C07196=1037.272,370.437,-131.137,172.942,44.628,158.763
C07197=1037.264,370.189,-131.097,172.935,44.625,158.762
C07198=1037.256,369.942,-131.057,172.928,44.622,158.760
C07199=1037.248,369.696,-131.017,172.921,44.619,158.759
C07200=1037.240,369.449,-130.977,172.914,44.615,158.757
C07201=1037.231,369.203,-130.937,172.907,44.612,158.756
C07202=1037.223,368.957,-130.897,172.900,44.608,158.754
C07203=1037.215,368.710,-130.857,172.894,44.605,158.753
C07204=1037.207,368.462,-130.817,172.887,44.602,158.751
C07205=1037.198,368.216,-130.778,172.881,44.599,158.750
C07206=1037.190,367.969,-130.739,172.874,44.595,158.748
C07207=1037.182,367.723,-130.698,172.867,44.592,158.747
C07208=1037.173,367.476,-130.659,172.860,44.589,158.745
C07209=1037.166,367.229,-130.619,172.853,44.586,158.744
C07210=1037.157,366.983,-130.579,172.848,44.582,158.743
C07211=1037.149,366.736,-130.539,172.841,44.579,158.741
C07212=1037.141,366.489,-130.500,172.834,44.576,158.740
C07213=1037.132,366.243,-130.461,172.827,44.573,158.738
C07214=1037.125,365.996,-130.421,172.820,44.570,158.737
C07215=1037.116,365.749,-130.382,172.814,44.566,158.735
C07216=1037.109,365.502,-130.342,172.807,44.563,158.734
C07217=1037.101,365.256,-130.303,172.801,44.560,158.733
C07218=1037.093,365.009,-130.263,172.794,44.557,158.731
C07219=1037.085,364.762,-130.224,172.788,44.554,158.730
C07220=1037.076,364.516,-130.185,172.781,44.551,158.728
C07221=1037.069,364.269,-130.145,172.774,44.548,158.727
C07222=1037.056,363.891,-130.084,172.765,44.543,158.725
C07223=1037.044,363.513,-130.025,172.755,44.538,158.723
C07224=1037.032,363.134,-129.964,172.745,44.533,158.721
C07225=1037.020,362.756,-129.904,172.735,44.528,158.719
C07226=1037.012,362.510,-129.865,172.729,44.525,158.717
C07227=1037.004,362.262,-129.826,172.722,44.522,158.716
C07228=1036.996,362.015,-129.786,172.716,44.519,158.715
C07229=1036.988,361.769,-129.748,172.710,44.516,158.713
C07230=1036.981,361.522,-129.708,172.703,44.513,158.712
C07231=1036.972,361.275,-129.669,172.697,44.510,158.711
C07232=1036.964,361.028,-129.630,172.690,44.508,158.709
C07233=1036.956,360.782,-129.592,172.685,44.504,158.708
C07234=1036.948,360.534,-129.553,172.678,44.501,158.707
C07235=1036.940,360.288,-129.514,172.671,44.499,158.705
C07236=1036.932,360.041,-129.476,172.666,44.495,158.704
C07237=1036.925,359.794,-129.437,172.659,44.493,158.703
C07238=1036.916,359.547,-129.397,172.653,44.490,158.701
C07239=1036.909,359.301,-129.359,172.647,44.486,158.700
C07240=1036.901,359.053,-129.320,172.640,44.484,158.699
C07241=1036.893,358.806,-129.282,172.634,44.481,158.698
C07242=1036.885,358.560,-129.243,172.628,44.478,158.696
C07243=1036.877,358.313,-129.204,172.622,44.475,158.695
C07244=1036.868,358.066,-129.166,172.615,44.472,158.694
C07245=1036.861,357.819,-129.127,172.610,44.470,158.693
C07246=1036.853,357.572,-129.089,172.603,44.467,158.691
C07247=1036.845,357.326,-129.050,172.598,44.464,158.690
C07248=1036.837,357.078,-129.012,172.591,44.461,158.689
C07249=1036.830,356.832,-128.973,172.585,44.458,158.687
C07250=1036.822,356.584,-128.934,172.579,44.456,158.686
C07251=1036.814,356.338,-128.896,172.573,44.453,158.685
C07252=1036.806,356.091,-128.858,172.566,44.450,158.684
C07253=1036.799,355.844,-128.819,172.561,44.447,158.682
C07254=1036.791,355.596,-128.781,172.554,44.444,158.681
C07255=1036.783,355.350,-128.744,172.549,44.442,158.680
C07256=1036.774,355.103,-128.705,172.542,44.439,158.679
C07257=1036.767,354.856,-128.667,172.537,44.437,158.678
C07258=1036.759,354.609,-128.629,172.530,44.434,158.676
C07259=1036.752,354.362,-128.591,172.524,44.431,158.675
C07260=1036.743,354.115,-128.552,172.518,44.428,158.674
C07261=1036.736,353.868,-128.515,172.512,44.425,158.673
C07262=1036.729,353.621,-128.476,172.507,44.423,158.672
C07263=1036.720,353.374,-128.438,172.500,44.420,158.670
C07264=1036.712,353.127,-128.401,172.495,44.417,158.669
C07265=1036.704,352.880,-128.362,172.488,44.415,158.668
C07266=1036.697,352.633,-128.324,172.483,44.412,158.667
C07267=1036.689,352.386,-128.286,172.476,44.410,158.666
C07268=1036.681,352.139,-128.248,172.471,44.407,158.664
C07269=1036.674,351.892,-128.210,172.465,44.404,158.663
C07270=1036.666,351.646,-128.173,172.459,44.402,158.662
C07271=1036.659,351.399,-128.135,172.454,44.400,158.661
C07272=1036.651,351.151,-128.097,172.448,44.397,158.660
C07273=1036.643,350.904,-128.059,172.441,44.394,158.659
C07274=1036.636,350.657,-128.022,172.436,44.391,158.657
C07275=1036.628,350.410,-127.983,172.430,44.389,158.656
C07276=1036.620,350.163,-127.946,172.424,44.387,158.655
C07277=1036.613,349.916,-127.908,172.419,44.384,158.654
C07278=1036.601,349.544,-127.851,172.409,44.380,158.652
C07279=1036.590,349.171,-127.795,172.401,44.376,158.651
C07280=1036.578,348.799,-127.738,172.392,44.373,158.649
C07281=1036.567,348.427,-127.682,172.384,44.369,158.647
C07282=1036.559,348.180,-127.645,172.379,44.366,158.646
C07283=1036.552,347.933,-127.607,172.372,44.364,158.645
C07284=1036.543,347.686,-127.570,172.367,44.362,158.644
C07285=1036.536,347.439,-127.533,172.361,44.359,158.643
C07286=1036.529,347.192,-127.495,172.355,44.357,158.642
C07287=1036.521,346.945,-127.458,172.350,44.354,158.641
C07288=1036.513,346.698,-127.421,172.344,44.352,158.640
C07289=1036.505,346.451,-127.384,172.339,44.349,158.638
C07290=1036.498,346.204,-127.346,172.332,44.347,158.637
C07291=1036.491,345.956,-127.309,172.327,44.345,158.636
C07292=1036.483,345.710,-127.272,172.322,44.343,158.635
C07293=1036.475,345.462,-127.234,172.316,44.340,158.634
C07294=1036.467,345.215,-127.197,172.310,44.338,158.633
C07295=1036.460,344.968,-127.159,172.305,44.336,158.632
C07296=1036.452,344.720,-127.123,172.299,44.333,158.631
C07297=1036.445,344.473,-127.086,172.294,44.331,158.630
C07298=1036.437,344.226,-127.049,172.289,44.329,158.629
C07299=1036.430,343.979,-127.011,172.282,44.326,158.628
C07300=1036.422,343.732,-126.975,172.277,44.324,158.627
C07301=1036.415,343.485,-126.937,172.272,44.322,158.626
C07302=1036.407,343.238,-126.901,172.266,44.320,158.625
C07303=1036.400,342.991,-126.864,172.261,44.317,158.623
C07304=1036.392,342.744,-126.827,172.256,44.315,158.622
C07305=1036.385,342.497,-126.790,172.249,44.313,158.621
C07306=1036.378,342.249,-126.753,172.244,44.310,158.620
C07307=1036.370,342.002,-126.716,172.239,44.308,158.619
C07308=1036.363,341.755,-126.680,172.233,44.306,158.618
C07309=1036.355,341.508,-126.642,172.228,44.303,158.617
C07310=1036.348,341.260,-126.606,172.223,44.301,158.616
C07311=1036.340,341.013,-126.569,172.218,44.299,158.615
C07312=1036.333,340.766,-126.532,172.211,44.297,158.614
C07313=1036.325,340.518,-126.496,172.206,44.295,158.613
C07314=1036.318,340.272,-126.459,172.201,44.293,158.612
C07315=1036.310,340.025,-126.423,172.196,44.291,158.611
C07316=1036.303,339.777,-126.386,172.190,44.288,158.610
C07317=1036.295,339.530,-126.349,172.185,44.286,158.609
C07318=1036.287,339.283,-126.313,172.180,44.284,158.608
C07319=1036.280,339.035,-126.277,172.175,44.282,158.607
C07320=1036.273,338.788,-126.241,172.168,44.280,158.606
C07321=1036.265,338.541,-126.204,172.163,44.278,158.605
C07322=1036.258,338.294,-126.167,172.158,44.275,158.604
C07323=1036.250,338.046,-126.131,172.153,44.273,158.603
C07324=1036.243,337.800,-126.095,172.148,44.272,158.602
C07325=1036.236,337.552,-126.059,172.142,44.270,158.601
C07326=1036.228,337.304,-126.022,172.137,44.267,158.600
C07327=1036.221,337.057,-125.986,172.132,44.265,158.599
C07328=1036.214,336.810,-125.950,172.127,44.263,158.598
C07329=1036.206,336.563,-125.913,172.121,44.261,158.597
C07330=1036.199,336.316,-125.876,172.116,44.259,158.597
C07331=1036.192,336.069,-125.841,172.111,44.257,158.596
C07332=1036.184,335.822,-125.804,172.106,44.255,158.595
C07333=1036.176,335.574,-125.768,172.101,44.253,158.594
C07334=1036.165,335.199,-125.713,172.093,44.250,158.592
C07335=1036.154,334.823,-125.659,172.085,44.247,158.591
C07336=1036.143,334.447,-125.604,172.077,44.244,158.589
C07337=1036.132,334.071,-125.550,172.070,44.241,158.588
C07338=1036.125,333.824,-125.513,172.064,44.238,158.587
C07339=1036.118,333.577,-125.478,172.059,44.237,158.586
C07340=1036.110,333.330,-125.441,172.054,44.235,158.585
C07341=1036.103,333.082,-125.406,172.049,44.233,158.584
C07342=1036.095,332.835,-125.370,172.044,44.231,158.583
C07343=1036.088,332.588,-125.334,172.039,44.229,158.583
C07344=1036.081,332.340,-125.299,172.034,44.227,158.582
C07345=1036.073,332.093,-125.262,172.029,44.226,158.581
C07346=1036.066,331.846,-125.227,172.023,44.223,158.580
C07347=1036.058,331.598,-125.192,172.018,44.222,158.579
C07348=1036.051,331.351,-125.156,172.013,44.220,158.578
C07349=1036.044,331.103,-125.120,172.008,44.218,158.577
C07350=1036.037,330.857,-125.084,172.003,44.216,158.576
C07351=1036.029,330.609,-125.049,171.998,44.214,158.575
C07352=1036.022,330.362,-125.013,171.993,44.213,158.574
C07353=1036.015,330.114,-124.978,171.988,44.210,158.573
C07354=1036.008,329.867,-124.942,171.983,44.209,158.573
C07355=1036.000,329.619,-124.906,171.978,44.207,158.572
C07356=1035.993,329.372,-124.870,171.973,44.205,158.571
C07357=1035.986,329.124,-124.835,171.968,44.203,158.570
C07358=1035.979,328.877,-124.799,171.963,44.202,158.569
C07359=1035.972,328.630,-124.764,171.958,44.199,158.568
C07360=1035.965,328.382,-124.728,171.953,44.198,158.567
C07361=1035.957,328.136,-124.693,171.948,44.196,158.567
C07362=1035.950,327.888,-124.658,171.943,44.195,158.566
C07363=1035.942,327.640,-124.623,171.938,44.193,158.565
C07364=1035.935,327.392,-124.588,171.933,44.191,158.564
C07365=1035.927,327.145,-124.553,171.928,44.189,158.563
C07366=1035.920,326.898,-124.518,171.924,44.187,158.562
C07367=1035.912,326.651,-124.482,171.919,44.186,158.562
C07368=1035.905,326.403,-124.447,171.914,44.184,158.561
C07369=1035.897,326.156,-124.412,171.909,44.183,158.560
C07370=1035.890,325.908,-124.377,171.904,44.181,158.559
C07371=1035.883,325.661,-124.343,171.899,44.179,158.558
C07372=1035.875,325.413,-124.307,171.894,44.178,158.557
C07373=1035.868,325.166,-124.273,171.890,44.176,158.557
C07374=1035.861,324.919,-124.237,171.885,44.174,158.556
C07375=1035.853,324.671,-124.202,171.880,44.173,158.555
C07376=1035.846,324.424,-124.167,171.875,44.171,158.554
C07377=1035.839,324.177,-124.133,171.870,44.169,158.553
C07378=1035.831,323.929,-124.097,171.865,44.168,158.553
C07379=1035.824,323.682,-124.063,171.860,44.166,158.552
C07380=1035.817,323.434,-124.028,171.856,44.164,158.551
C07381=1035.810,323.186,-123.994,171.851,44.163,158.550
C07382=1035.803,322.938,-123.958,171.846,44.161,158.549
C07383=1035.795,322.691,-123.924,171.841,44.160,158.549
C07384=1035.788,322.444,-123.889,171.836,44.159,158.548
C07385=1035.781,322.197,-123.854,171.832,44.157,158.547
C07386=1035.774,321.950,-123.819,171.827,44.155,158.546
C07387=1035.766,321.701,-123.785,171.822,44.153,158.545
C07388=1035.759,321.454,-123.750,171.817,44.152,158.545
C07389=1035.752,321.207,-123.715,171.813,44.150,158.544
C07390=1035.741,320.826,-123.661,171.806,44.148,158.543
C07391=1035.730,320.447,-123.609,171.799,44.146,158.541
C07392=1035.719,320.066,-123.556,171.791,44.143,158.540
C07393=1035.709,319.685,-123.502,171.785,44.141,158.539
C07394=1035.701,319.438,-123.468,171.780,44.139,158.538
C07395=1035.694,319.191,-123.434,171.775,44.138,158.538
C07396=1035.687,318.943,-123.399,171.770,44.137,158.537
C07397=1035.680,318.696,-123.364,171.766,44.135,158.536
C07398=1035.673,318.448,-123.330,171.761,44.133,158.535
C07399=1035.666,318.201,-123.295,171.756,44.132,158.534
C07400=1035.659,317.953,-123.261,171.752,44.130,158.534
C07401=1035.652,317.706,-123.226,171.747,44.129,158.533
C07402=1035.645,317.458,-123.192,171.742,44.128,158.532
C07403=1035.638,317.211,-123.157,171.738,44.126,158.531
C07404=1035.631,316.963,-123.123,171.733,44.124,158.531
C07405=1035.624,316.716,-123.088,171.729,44.123,158.530
C07406=1035.617,316.468,-123.054,171.725,44.121,158.529
C07407=1035.610,316.221,-123.019,171.720,44.120,158.528
C07408=1035.603,315.973,-122.985,171.715,44.119,158.528
C07409=1035.596,315.725,-122.951,171.711,44.117,158.527
C07410=1035.589,315.478,-122.917,171.706,44.116,158.526
C07411=1035.581,315.231,-122.883,171.701,44.114,158.525
C07412=1035.575,314.983,-122.848,171.697,44.112,158.525
C07413=1035.567,314.736,-122.814,171.692,44.111,158.524
C07414=1035.562,314.488,-122.780,171.687,44.110,158.523
C07415=1035.554,314.241,-122.746,171.684,44.108,158.523
C07416=1035.548,313.993,-122.711,171.679,44.107,158.522
C07417=1035.540,313.746,-122.677,171.675,44.106,158.521
C07418=1035.533,313.498,-122.643,171.670,44.104,158.520
C07419=1035.527,313.250,-122.609,171.665,44.103,158.520
C07420=1035.520,313.004,-122.574,171.661,44.101,158.519
C07421=1035.513,312.756,-122.540,171.657,44.100,158.518
C07422=1035.506,312.508,-122.506,171.653,44.098,158.517
C07423=1035.499,312.260,-122.472,171.648,44.097,158.517
C07424=1035.493,312.012,-122.438,171.643,44.096,158.516
C07425=1035.486,311.765,-122.405,171.639,44.094,158.515
C07426=1035.479,311.518,-122.371,171.634,44.093,158.515
C07427=1035.472,311.270,-122.337,171.630,44.091,158.514
C07428=1035.464,311.022,-122.303,171.626,44.090,158.513
C07429=1035.457,310.775,-122.269,171.621,44.089,158.513
C07430=1035.450,310.527,-122.235,171.617,44.088,158.512
C07431=1035.443,310.280,-122.203,171.612,44.087,158.511
C07432=1035.435,310.033,-122.169,171.608,44.085,158.511
C07433=1035.428,309.785,-122.135,171.604,44.084,158.510
C07434=1035.421,309.537,-122.102,171.599,44.083,158.509
C07435=1035.414,309.289,-122.068,171.595,44.082,158.509
C07436=1035.407,309.042,-122.035,171.590,44.080,158.508
C07437=1035.400,308.795,-122.001,171.586,44.079,158.507
C07438=1035.393,308.546,-121.968,171.582,44.078,158.507
C07439=1035.385,308.299,-121.934,171.577,44.077,158.506
C07440=1035.379,308.052,-121.901,171.573,44.076,158.505
C07441=1035.371,307.804,-121.868,171.568,44.075,158.505
C07442=1035.364,307.556,-121.835,171.565,44.074,158.504
C07443=1035.357,307.308,-121.801,171.560,44.073,158.503
C07444=1035.350,307.061,-121.767,171.556,44.071,158.503
C07445=1035.343,306.813,-121.734,171.551,44.070,158.502
C07446=1035.332,306.438,-121.684,171.545,44.068,158.501
C07447=1035.322,306.063,-121.633,171.538,44.066,158.500
C07448=1035.311,305.687,-121.582,171.532,44.065,158.499
C07449=1035.300,305.312,-121.533,171.526,44.063,158.498
C07450=1035.293,305.064,-121.499,171.521,44.062,158.497
C07451=1035.286,304.816,-121.466,171.517,44.061,158.497
C07452=1035.280,304.569,-121.433,171.512,44.060,158.496
C07453=1035.272,304.321,-121.399,171.509,44.058,158.496
C07454=1035.261,303.916,-121.345,171.501,44.057,158.495
C07455=1035.250,303.511,-121.291,171.494,44.055,158.493
C07456=1035.238,303.106,-121.237,171.487,44.053,158.493
C07457=1035.227,302.701,-121.183,171.481,44.051,158.492
C07458=1035.220,302.453,-121.150,171.476,44.050,158.491
C07459=1035.213,302.205,-121.117,171.473,44.049,158.490
C07460=1035.206,301.957,-121.083,171.468,44.048,158.490
C07461=1035.199,301.710,-121.051,171.464,44.047,158.489
C07462=1035.192,301.462,-121.018,171.459,44.046,158.488
C07463=1035.186,301.215,-120.984,171.456,44.045,158.488
C07464=1035.179,300.966,-120.951,171.452,44.043,158.487
C07465=1035.172,300.719,-120.919,171.447,44.043,158.487
C07466=1035.165,300.471,-120.886,171.444,44.042,158.486
C07467=1035.158,300.224,-120.853,171.439,44.041,158.485
C07468=1035.152,299.976,-120.820,171.435,44.039,158.485
C07469=1035.144,299.728,-120.787,171.430,44.038,158.484
C07470=1035.138,299.481,-120.755,171.427,44.037,158.483
C07471=1035.131,299.232,-120.722,171.423,44.036,158.483
C07472=1035.124,298.985,-120.688,171.418,44.035,158.482
C07473=1035.117,298.737,-120.656,171.415,44.034,158.482
C07474=1035.111,298.490,-120.623,171.410,44.033,158.481
C07475=1035.104,298.242,-120.590,171.406,44.032,158.481
C07476=1035.097,297.994,-120.557,171.402,44.031,158.480
C07477=1035.090,297.747,-120.525,171.398,44.030,158.479
C07478=1035.084,297.499,-120.492,171.394,44.029,158.479
C07479=1035.077,297.251,-120.459,171.390,44.028,158.478
C07480=1035.071,297.003,-120.426,171.386,44.027,158.478
C07481=1035.064,296.756,-120.394,171.382,44.026,158.477
C07482=1035.057,296.508,-120.361,171.378,44.025,158.476
C07483=1035.051,296.260,-120.328,171.374,44.024,158.476
C07484=1035.044,296.012,-120.295,171.370,44.022,158.475
C07485=1035.037,295.764,-120.263,171.366,44.022,158.475
C07486=1035.030,295.517,-120.230,171.362,44.021,158.474
C07487=1035.024,295.269,-120.197,171.358,44.019,158.473
C07488=1035.016,295.021,-120.165,171.354,44.018,158.473
C07489=1035.010,294.774,-120.132,171.350,44.018,158.472
C07490=1035.003,294.526,-120.100,171.346,44.017,158.472
C07491=1034.996,294.278,-120.067,171.341,44.016,158.471
C07492=1034.989,294.031,-120.035,171.338,44.015,158.471
C07493=1034.983,293.783,-120.003,171.334,44.014,158.470
C07494=1034.976,293.535,-119.970,171.329,44.013,158.470
C07495=1034.969,293.287,-119.938,171.326,44.013,158.469
C07496=1034.963,293.039,-119.906,171.322,44.011,158.469
C07497=1034.956,292.792,-119.874,171.318,44.011,158.468
C07498=1034.949,292.567,-119.844,171.314,44.010,158.467
C07499=1034.943,292.343,-119.815,171.311,44.009,158.467
C07500=1034.937,292.118,-119.786,171.307,44.008,158.467
C07501=1034.930,291.894,-119.757,171.304,44.008,158.466
C07502=1034.924,291.670,-119.728,171.300,44.006,158.465
C07503=1034.918,291.446,-119.699,171.296,44.006,158.465
C07504=1034.912,291.221,-119.670,171.293,44.005,158.465
C07505=1034.906,290.997,-119.640,171.289,44.005,158.464
C07506=1034.899,290.749,-119.609,171.286,44.003,158.463
C07507=1034.892,290.501,-119.576,171.282,44.003,158.463
C07508=1034.885,290.253,-119.545,171.277,44.002,158.462
C07509=1034.879,290.005,-119.512,171.274,44.001,158.462
C07510=1034.872,289.758,-119.481,171.270,44.000,158.461
C07511=1034.865,289.510,-119.449,171.267,43.999,158.461
C07512=1034.857,289.262,-119.417,171.262,43.999,158.460
C07513=1034.851,289.014,-119.384,171.259,43.998,158.460
C07514=1034.844,288.766,-119.353,171.255,43.997,158.459
C07515=1034.838,288.518,-119.321,171.250,43.996,158.459
C07516=1034.831,288.271,-119.289,171.247,43.996,158.458
C07517=1034.823,288.022,-119.257,171.243,43.994,158.458
C07518=1034.816,287.775,-119.225,171.240,43.994,158.457
C07519=1034.810,287.527,-119.193,171.235,43.993,158.457
C07520=1034.804,287.279,-119.162,171.231,43.992,158.456
C07521=1034.797,287.032,-119.130,171.228,43.991,158.456
C07522=1034.790,286.784,-119.098,171.224,43.991,158.455
C07523=1034.783,286.536,-119.067,171.220,43.990,158.455
C07524=1034.776,286.288,-119.035,171.216,43.989,158.454
C07525=1034.769,286.040,-119.003,171.213,43.988,158.454
C07526=1034.762,285.792,-118.971,171.209,43.988,158.453
C07527=1034.755,285.544,-118.940,171.205,43.987,158.453
C07528=1034.749,285.296,-118.908,171.201,43.986,158.452
C07529=1034.742,285.048,-118.877,171.197,43.985,158.452
C07530=1034.735,284.801,-118.846,171.194,43.985,158.451
C07531=1034.728,284.553,-118.813,171.189,43.984,158.451
C07532=1034.721,284.305,-118.782,171.186,43.984,158.450
C07533=1034.714,284.057,-118.750,171.182,43.983,158.450
C07534=1034.707,283.809,-118.719,171.179,43.982,158.449
C07535=1034.701,283.561,-118.687,171.174,43.981,158.449
C07536=1034.694,283.313,-118.656,171.171,43.981,158.448
C07537=1034.687,283.065,-118.624,171.167,43.980,158.448
C07538=1034.680,282.817,-118.593,171.164,43.979,158.447
C07539=1034.674,282.569,-118.562,171.160,43.979,158.447
C07540=1034.667,282.321,-118.530,171.156,43.978,158.447
C07541=1034.660,282.074,-118.499,171.152,43.978,158.446
C07542=1034.654,281.826,-118.467,171.148,43.976,158.445
C07543=1034.647,281.578,-118.436,171.145,43.976,158.445
C07544=1034.640,281.330,-118.404,171.141,43.975,158.445
C07545=1034.633,281.082,-118.373,171.137,43.975,158.444
C07546=1034.627,280.834,-118.342,171.133,43.974,158.444
C07547=1034.619,280.586,-118.311,171.130,43.973,158.443
C07548=1034.612,280.339,-118.279,171.126,43.973,158.443
C07549=1034.606,280.090,-118.249,171.123,43.972,158.442
C07550=1034.599,279.842,-118.217,171.119,43.972,158.442
C07551=1034.593,279.594,-118.186,171.115,43.971,158.441
C07552=1034.586,279.346,-118.154,171.111,43.970,158.441
C07553=1034.579,279.098,-118.123,171.108,43.970,158.440
C07554=1034.573,278.851,-118.092,171.104,43.969,158.440
C07555=1034.567,278.603,-118.061,171.101,43.968,158.440
C07556=1034.560,278.355,-118.030,171.097,43.968,158.439
C07557=1034.553,278.107,-117.998,171.094,43.967,158.439
C07558=1034.544,277.761,-117.955,171.088,43.966,158.438
C07559=1034.534,277.414,-117.912,171.083,43.965,158.437
C07560=1034.524,277.067,-117.869,171.078,43.965,158.437
C07561=1034.515,276.721,-117.825,171.073,43.964,158.436
C07562=1034.508,276.473,-117.794,171.070,43.963,158.436
C07563=1034.501,276.224,-117.763,171.066,43.963,158.435
C07564=1034.494,275.977,-117.732,171.063,43.962,158.435
C07565=1034.488,275.728,-117.701,171.058,43.962,158.434
C07566=1034.481,275.480,-117.670,171.055,43.961,158.434
C07567=1034.475,275.233,-117.640,171.051,43.961,158.434
C07568=1034.468,274.985,-117.609,171.048,43.960,158.433
C07569=1034.461,274.737,-117.577,171.044,43.960,158.433
C07570=1034.454,274.489,-117.547,171.041,43.959,158.432
C07571=1034.447,274.241,-117.516,171.037,43.958,158.432
C07572=1034.441,273.992,-117.485,171.034,43.958,158.431
C07573=1034.435,273.745,-117.455,171.030,43.957,158.431
C07574=1034.427,273.497,-117.424,171.027,43.957,158.431
C07575=1034.421,273.249,-117.393,171.023,43.956,158.430
C07576=1034.413,273.001,-117.362,171.019,43.956,158.430
C07577=1034.407,272.752,-117.332,171.016,43.955,158.429
C07578=1034.400,272.505,-117.300,171.012,43.955,158.429
C07579=1034.394,272.257,-117.271,171.009,43.954,158.428
C07580=1034.387,272.009,-117.240,171.005,43.954,158.428
C07581=1034.380,271.761,-117.209,171.002,43.953,158.428
C07582=1034.373,271.512,-117.178,170.998,43.953,158.427
C07583=1034.368,271.265,-117.148,170.995,43.953,158.427
C07584=1034.360,271.017,-117.117,170.992,43.952,158.426
C07585=1034.354,270.768,-117.086,170.988,43.951,158.426
C07586=1034.347,270.520,-117.056,170.985,43.951,158.425
C07587=1034.341,270.272,-117.026,170.981,43.951,158.425
C07588=1034.333,270.025,-116.995,170.978,43.950,158.425
C07589=1034.326,269.777,-116.965,170.973,43.949,158.424
C07590=1034.320,269.528,-116.934,170.970,43.949,158.424
C07591=1034.313,269.281,-116.904,170.967,43.949,158.423
C07592=1034.307,269.032,-116.874,170.963,43.948,158.423
C07593=1034.299,268.784,-116.843,170.960,43.948,158.423
C07594=1034.293,268.536,-116.812,170.956,43.947,158.422
C07595=1034.286,268.288,-116.782,170.953,43.947,158.422
C07596=1034.279,268.040,-116.752,170.950,43.947,158.422
C07597=1034.273,267.792,-116.722,170.946,43.946,158.421
C07598=1034.266,267.544,-116.692,170.943,43.945,158.421
C07599=1034.260,267.296,-116.661,170.939,43.945,158.420
C07600=1034.253,267.047,-116.631,170.936,43.945,158.420
C07601=1034.246,266.800,-116.600,170.932,43.945,158.420
C07602=1034.239,266.552,-116.570,170.929,43.944,158.419
C07603=1034.232,266.304,-116.540,170.926,43.943,158.419
C07604=1034.225,266.056,-116.510,170.922,43.943,158.418
C07605=1034.219,265.807,-116.480,170.919,43.943,158.418
C07606=1034.212,265.559,-116.450,170.915,43.943,158.418
C07607=1034.205,265.311,-116.420,170.912,43.942,158.417
C07608=1034.199,265.063,-116.390,170.909,43.942,158.417
C07609=1034.192,264.815,-116.359,170.905,43.941,158.416
C07610=1034.186,264.567,-116.329,170.902,43.941,158.416
C07611=1034.178,264.319,-116.299,170.898,43.941,158.416
C07612=1034.172,264.070,-116.269,170.895,43.941,158.415
C07613=1034.165,263.823,-116.239,170.892,43.940,158.415
C07614=1034.156,263.481,-116.197,170.887,43.939,158.415
C07615=1034.147,263.139,-116.156,170.883,43.939,158.414
C07616=1034.138,262.798,-116.115,170.878,43.939,158.414
C07617=1034.129,262.455,-116.074,170.874,43.938,158.413
C07618=1034.122,262.207,-116.044,170.870,43.937,158.413
C07619=1034.115,261.959,-116.014,170.867,43.937,158.412
C07620=1034.109,261.711,-115.983,170.863,43.937,158.412
C07621=1034.102,261.463,-115.953,170.860,43.937,158.412
C07622=1034.095,261.215,-115.924,170.857,43.936,158.411
C07623=1034.088,260.966,-115.894,170.853,43.936,158.411
C07624=1034.081,260.718,-115.865,170.850,43.936,158.411
C07625=1034.074,260.470,-115.835,170.847,43.935,158.410
C07626=1034.067,260.222,-115.805,170.843,43.935,158.410
C07627=1034.061,259.974,-115.776,170.840,43.935,158.409
C07628=1034.053,259.726,-115.746,170.837,43.935,158.409
C07629=1034.047,259.478,-115.717,170.833,43.935,158.409
C07630=1034.040,259.229,-115.687,170.830,43.935,158.408
C07631=1034.033,258.981,-115.658,170.827,43.934,158.408
C07632=1034.026,258.733,-115.628,170.823,43.934,158.408
C07633=1034.019,258.484,-115.599,170.820,43.934,158.407
C07634=1034.013,258.237,-115.569,170.817,43.934,158.407
C07635=1034.006,257.988,-115.540,170.813,43.933,158.407
C07636=1033.999,257.741,-115.510,170.810,43.933,158.406
C07637=1033.992,257.492,-115.481,170.807,43.933,158.406
C07638=1033.986,257.244,-115.451,170.803,43.933,158.406
C07639=1033.979,256.995,-115.421,170.800,43.932,158.405
C07640=1033.972,256.748,-115.392,170.797,43.932,158.405
C07641=1033.965,256.499,-115.363,170.793,43.932,158.405
C07642=1033.958,256.251,-115.334,170.790,43.932,158.404
C07643=1033.951,256.003,-115.304,170.788,43.931,158.404
C07644=1033.945,255.755,-115.275,170.784,43.931,158.404
C07645=1033.938,255.507,-115.245,170.781,43.931,158.404
C07646=1033.932,255.259,-115.216,170.778,43.931,158.403
C07647=1033.924,255.010,-115.187,170.774,43.931,158.403
C07648=1033.917,254.763,-115.157,170.771,43.931,158.402
C07649=1033.911,254.514,-115.128,170.768,43.930,158.402
C07650=1033.904,254.266,-115.099,170.765,43.930,158.402
C07651=1033.898,254.018,-115.069,170.761,43.930,158.401
C07652=1033.891,253.769,-115.039,170.758,43.930,158.401
C07653=1033.884,253.521,-115.011,170.755,43.930,158.401
C07654=1033.877,253.273,-114.982,170.752,43.929,158.401
C07655=1033.871,253.025,-114.952,170.749,43.929,158.400
C07656=1033.864,252.776,-114.922,170.746,43.929,158.400
C07657=1033.857,252.528,-114.893,170.742,43.929,158.400
C07658=1033.851,252.280,-114.864,170.739,43.929,158.399
C07659=1033.843,252.032,-114.835,170.736,43.929,158.399
C07660=1033.837,251.784,-114.806,170.732,43.928,158.399
C07661=1033.831,251.536,-114.777,170.730,43.928,158.398
C07662=1033.824,251.287,-114.747,170.727,43.928,158.398
C07663=1033.818,251.039,-114.718,170.723,43.928,158.398
C07664=1033.811,250.791,-114.688,170.720,43.928,158.397
C07665=1033.804,250.543,-114.660,170.717,43.927,158.397
C07666=1033.797,250.295,-114.631,170.713,43.927,158.397
C07667=1033.791,250.047,-114.602,170.710,43.927,158.396
C07668=1033.784,249.798,-114.572,170.708,43.927,158.396
C07669=1033.778,249.550,-114.543,170.705,43.927,158.396
C07670=1033.768,249.207,-114.502,170.700,43.926,158.395
C07671=1033.760,248.864,-114.462,170.696,43.926,158.395
C07672=1033.750,248.520,-114.422,170.691,43.926,158.395
C07673=1033.741,248.177,-114.382,170.687,43.925,158.394
C07674=1033.735,247.929,-114.353,170.684,43.925,158.394
C07675=1033.728,247.680,-114.324,170.681,43.925,158.394
C07676=1033.722,247.432,-114.295,170.678,43.925,158.393
C07677=1033.715,247.184,-114.266,170.675,43.925,158.393
C07678=1033.709,246.936,-114.237,170.671,43.924,158.392
C07679=1033.702,246.687,-114.208,170.668,43.924,158.392
C07680=1033.696,246.439,-114.179,170.666,43.924,158.392
C07681=1033.689,246.191,-114.150,170.663,43.924,158.392
C07682=1033.682,245.943,-114.121,170.659,43.924,158.391
C07683=1033.676,245.694,-114.092,170.656,43.924,158.391
C07684=1033.669,245.446,-114.063,170.654,43.924,158.391
C07685=1033.663,245.198,-114.034,170.650,43.923,158.390
C07686=1033.657,244.950,-114.005,170.647,43.923,158.390
C07687=1033.650,244.702,-113.976,170.644,43.923,158.390
C07688=1033.643,244.452,-113.948,170.641,43.923,158.390
C07689=1033.637,244.204,-113.919,170.638,43.923,158.389
C07690=1033.630,243.956,-113.890,170.635,43.923,158.389
C07691=1033.624,243.708,-113.861,170.632,43.923,158.389
C07692=1033.617,243.461,-113.833,170.628,43.923,158.388
C07693=1033.610,243.211,-113.804,170.626,43.922,158.388
C07694=1033.603,242.963,-113.776,170.623,43.922,158.388
C07695=1033.597,242.715,-113.747,170.620,43.922,158.388
C07696=1033.590,242.467,-113.718,170.616,43.922,158.387
C07697=1033.584,242.219,-113.690,170.614,43.922,158.387
C07698=1033.577,241.970,-113.661,170.611,43.922,158.387
C07699=1033.570,241.722,-113.632,170.608,43.922,158.386
C07700=1033.564,241.473,-113.604,170.604,43.922,158.386
C07701=1033.557,241.225,-113.575,170.602,43.922,158.386
C07702=1033.550,240.977,-113.547,170.599,43.922,158.386
C07703=1033.544,240.729,-113.518,170.596,43.922,158.385
C07704=1033.537,240.481,-113.490,170.592,43.921,158.385
C07705=1033.531,240.232,-113.461,170.590,43.921,158.385
C07706=1033.524,239.984,-113.433,170.587,43.921,158.384
C07707=1033.517,239.736,-113.404,170.583,43.921,158.384
C07708=1033.511,239.487,-113.376,170.580,43.922,158.384
C07709=1033.504,239.239,-113.348,170.578,43.922,158.384
C07710=1033.497,238.991,-113.320,170.575,43.921,158.383
C07711=1033.490,238.742,-113.290,170.572,43.921,158.383
C07712=1033.484,238.494,-113.263,170.568,43.921,158.383
C07713=1033.477,238.246,-113.234,170.566,43.921,158.383
C07714=1033.470,237.997,-113.207,170.563,43.921,158.382
C07715=1033.464,237.749,-113.177,170.560,43.921,158.382
C07716=1033.457,237.501,-113.150,170.557,43.922,158.382
C07717=1033.450,237.253,-113.121,170.554,43.921,158.382
C07718=1033.443,237.004,-113.094,170.551,43.921,158.381
C07719=1033.438,236.756,-113.065,170.548,43.921,158.381
C07720=1033.430,236.507,-113.036,170.544,43.921,158.381
C07721=1033.423,236.259,-113.009,170.542,43.921,158.381
C07722=1033.416,236.011,-112.980,170.539,43.922,158.380
C07723=1033.410,235.762,-112.953,170.536,43.922,158.380
C07724=1033.404,235.514,-112.924,170.534,43.921,158.380
C07725=1033.397,235.266,-112.896,170.530,43.921,158.380
C07726=1033.387,234.916,-112.856,170.526,43.921,158.379
C07727=1033.378,234.568,-112.817,170.522,43.922,158.379
C07728=1033.368,234.218,-112.778,170.519,43.922,158.379
C07729=1033.359,233.869,-112.738,170.514,43.922,158.378
C07730=1033.352,233.620,-112.710,170.511,43.922,158.378
C07731=1033.346,233.372,-112.682,170.508,43.922,158.378
C07732=1033.339,233.123,-112.654,170.506,43.921,158.377
C07733=1033.332,232.875,-112.626,170.502,43.921,158.377
C07734=1033.326,232.627,-112.598,170.499,43.922,158.377
C07735=1033.319,232.378,-112.570,170.497,43.922,158.377
C07736=1033.313,232.130,-112.542,170.494,43.922,158.376
C07737=1033.306,231.882,-112.513,170.490,43.922,158.376
C07738=1033.299,231.633,-112.486,170.488,43.922,158.376
C07739=1033.293,231.385,-112.458,170.485,43.922,158.376
C07740=1033.286,231.137,-112.430,170.482,43.922,158.376
C07741=1033.279,230.888,-112.402,170.480,43.922,158.375
C07742=1033.273,230.640,-112.375,170.477,43.922,158.375
C07743=1033.267,230.392,-112.347,170.473,43.922,158.375
C07744=1033.260,230.144,-112.319,170.471,43.922,158.375
C07745=1033.253,229.896,-112.291,170.468,43.922,158.374
C07746=1033.246,229.647,-112.263,170.465,43.922,158.374
C07747=1033.240,229.399,-112.236,170.463,43.922,158.374
C07748=1033.233,229.150,-112.208,170.459,43.922,158.374
C07749=1033.227,228.902,-112.180,170.456,43.923,158.373
C07750=1033.220,228.653,-112.152,170.454,43.923,158.373
C07751=1033.214,228.405,-112.124,170.451,43.923,158.373
C07752=1033.207,228.156,-112.096,170.448,43.922,158.373
C07753=1033.200,227.908,-112.069,170.445,43.923,158.373
C07754=1033.193,227.660,-112.042,170.442,43.923,158.372
C07755=1033.186,227.411,-112.014,170.440,43.923,158.372
C07756=1033.179,227.163,-111.986,170.437,43.923,158.372
C07757=1033.173,226.914,-111.958,170.434,43.923,158.372
C07758=1033.166,226.666,-111.931,170.432,43.923,158.371
C07759=1033.160,226.417,-111.904,170.428,43.923,158.371
C07760=1033.153,226.169,-111.877,170.425,43.923,158.371
C07761=1033.146,225.921,-111.849,170.423,43.924,158.371
C07762=1033.140,225.673,-111.821,170.420,43.924,158.371
C07763=1033.133,225.424,-111.794,170.418,43.924,158.370
C07764=1033.126,225.176,-111.766,170.414,43.924,158.370
C07765=1033.119,224.928,-111.739,170.411,43.925,158.370
C07766=1033.112,224.679,-111.712,170.409,43.924,158.370
C07767=1033.106,224.430,-111.684,170.406,43.924,158.369
C07768=1033.099,224.182,-111.656,170.403,43.925,158.369
C07769=1033.092,223.933,-111.629,170.401,43.925,158.369
C07770=1033.086,223.686,-111.602,170.398,43.925,158.369
C07771=1033.079,223.437,-111.575,170.395,43.925,158.369
C07772=1033.072,223.188,-111.547,170.392,43.925,158.368
C07773=1033.066,222.940,-111.519,170.389,43.926,158.368
C07774=1033.059,222.691,-111.492,170.387,43.925,158.368
C07775=1033.052,222.443,-111.465,170.384,43.926,158.368
C07776=1033.045,222.194,-111.438,170.381,43.926,158.368
C07777=1033.039,221.946,-111.410,170.378,43.926,158.367
C07778=1033.033,221.697,-111.383,170.375,43.926,158.367
C07779=1033.025,221.449,-111.356,170.373,43.926,158.367
C07780=1033.019,221.201,-111.328,170.370,43.927,158.367
C07781=1033.012,220.952,-111.301,170.368,43.926,158.367
C07782=1033.003,220.596,-111.261,170.363,43.926,158.366
C07783=1032.993,220.239,-111.222,170.359,43.927,158.366
C07784=1032.984,219.883,-111.183,170.356,43.927,158.366
C07785=1032.975,219.526,-111.144,170.352,43.927,158.365
C07786=1032.968,219.277,-111.118,170.348,43.927,158.365
C07787=1032.961,219.028,-111.090,170.346,43.928,158.365
C07788=1032.954,218.780,-111.064,170.343,43.928,158.365
C07789=1032.947,218.531,-111.036,170.341,43.928,158.365
C07790=1032.941,218.283,-111.010,170.338,43.929,158.364
C07791=1032.934,218.035,-110.982,170.336,43.928,158.364
C07792=1032.927,217.786,-110.956,170.333,43.929,158.364
C07793=1032.920,217.538,-110.928,170.330,43.929,158.364
C07794=1032.913,217.289,-110.902,170.328,43.929,158.364
C07795=1032.907,217.041,-110.874,170.324,43.929,158.363
C07796=1032.900,216.792,-110.848,170.322,43.930,158.363
C07797=1032.893,216.544,-110.820,170.319,43.930,158.363
C07798=1032.886,216.295,-110.794,170.317,43.930,158.363
C07799=1032.880,216.047,-110.766,170.314,43.931,158.363
C07800=1032.873,215.799,-110.740,170.312,43.930,158.363
C07801=1032.867,215.550,-110.713,170.309,43.931,158.362
C07802=1032.859,215.301,-110.686,170.306,43.931,158.362
C07803=1032.854,215.053,-110.659,170.303,43.931,158.362
C07804=1032.846,214.805,-110.632,170.300,43.932,158.362
C07805=1032.840,214.556,-110.605,170.298,43.932,158.362
C07806=1032.833,214.308,-110.579,170.295,43.932,158.361
C07807=1032.827,214.059,-110.551,170.293,43.932,158.361
C07808=1032.819,213.811,-110.525,170.290,43.933,158.361
C07809=1032.813,213.562,-110.498,170.287,43.932,158.361
C07810=1032.806,213.314,-110.471,170.284,43.933,158.361
C07811=1032.800,213.065,-110.444,170.282,43.933,158.360
C07812=1032.793,212.816,-110.418,170.279,43.933,158.360
C07813=1032.787,212.569,-110.390,170.277,43.934,158.360
C07814=1032.780,212.320,-110.364,170.274,43.934,158.360
C07815=1032.773,212.071,-110.337,170.272,43.934,158.360
C07816=1032.767,211.823,-110.311,170.268,43.934,158.360
C07817=1032.760,211.574,-110.283,170.266,43.934,158.359
C07818=1032.753,211.326,-110.257,170.263,43.934,158.359
C07819=1032.747,211.077,-110.230,170.261,43.935,158.359
C07820=1032.740,210.828,-110.203,170.258,43.935,158.359
C07821=1032.733,210.580,-110.177,170.256,43.935,158.359
C07822=1032.727,210.332,-110.150,170.253,43.936,158.359
C07823=1032.720,210.083,-110.123,170.251,43.936,158.358
C07824=1032.713,209.835,-110.097,170.248,43.936,158.358
C07825=1032.707,209.586,-110.070,170.246,43.936,158.358
C07826=1032.700,209.337,-110.044,170.242,43.937,158.358
C07827=1032.693,209.089,-110.018,170.240,43.937,158.358
C07828=1032.687,208.840,-109.991,170.237,43.937,158.358
C07829=1032.680,208.593,-109.964,170.235,43.938,158.357
C07830=1032.673,208.344,-109.938,170.233,43.937,158.357
C07831=1032.666,208.095,-109.911,170.230,43.938,158.357
C07832=1032.660,207.847,-109.884,170.228,43.938,158.357
C07833=1032.653,207.598,-109.858,170.225,43.938,158.357
C07834=1032.646,207.350,-109.832,170.223,43.939,158.357
C07835=1032.639,207.101,-109.806,170.220,43.939,158.356
C07836=1032.632,206.853,-109.779,170.217,43.939,158.356
C07837=1032.626,206.604,-109.752,170.214,43.940,158.356
C07838=1032.617,206.253,-109.716,170.211,43.940,158.356
C07839=1032.606,205.902,-109.678,170.207,43.940,158.356
C07840=1032.597,205.551,-109.641,170.204,43.941,158.355
C07841=1032.588,205.200,-109.604,170.200,43.942,158.355
C07842=1032.562,204.151,-109.499,169.861,43.837,158.304
C07843=1032.556,203.902,-109.473,169.857,43.838,158.304
C07844=1032.550,203.653,-109.449,169.853,43.839,158.304
C07845=1032.544,203.405,-109.424,169.850,43.840,158.304
C07846=1032.537,203.157,-109.399,169.846,43.842,158.304
C07847=1032.531,202.907,-109.374,169.842,43.842,158.304
C07848=1032.525,202.659,-109.349,169.839,43.844,158.304
C07849=1032.519,202.411,-109.324,169.835,43.844,158.304
C07850=1032.514,202.161,-109.299,169.832,43.846,158.304
C07851=1032.507,201.913,-109.274,169.828,43.847,158.304
C07852=1032.501,201.664,-109.249,169.825,43.848,158.303
C07853=1032.495,201.416,-109.225,169.822,43.849,158.303
C07854=1032.489,201.167,-109.200,169.817,43.850,158.303
C07855=1032.483,200.918,-109.175,169.815,43.851,158.303
C07856=1032.477,200.669,-109.150,169.811,43.852,158.303
C07857=1032.472,200.421,-109.125,169.808,43.853,158.303
C07858=1032.465,200.172,-109.101,169.804,43.854,158.303
C07859=1032.459,199.923,-109.076,169.800,43.856,158.303
C07860=1032.452,199.675,-109.051,169.797,43.857,158.303
C07861=1032.446,199.426,-109.027,169.794,43.858,158.303
C07862=1032.440,199.177,-109.003,169.790,43.859,158.303
C07863=1032.434,198.928,-108.978,169.787,43.860,158.303
C07864=1032.427,198.679,-108.954,169.783,43.862,158.303
C07865=1032.422,198.431,-108.929,169.780,43.863,158.303
C07866=1032.415,198.182,-108.905,169.776,43.865,158.303
C07867=1032.409,197.933,-108.880,169.773,43.865,158.302
C07868=1032.403,197.685,-108.856,169.769,43.867,158.302
C07869=1032.397,197.436,-108.831,169.765,43.868,158.302
C07870=1032.390,197.187,-108.807,169.763,43.869,158.302
C07871=1032.384,196.938,-108.782,169.759,43.871,158.302
C07872=1032.378,196.690,-108.758,169.756,43.872,158.302
C07873=1032.372,196.441,-108.733,169.752,43.873,158.302
C07874=1032.365,196.192,-108.709,169.749,43.874,158.302
C07875=1032.360,195.943,-108.685,169.745,43.875,158.302
C07876=1032.353,195.695,-108.660,169.741,43.877,158.302
C07877=1032.348,195.446,-108.636,169.739,43.878,158.302
C07878=1032.341,195.197,-108.612,169.735,43.879,158.302
C07879=1032.335,194.948,-108.587,169.732,43.880,158.302
C07880=1032.329,194.701,-108.563,169.728,43.882,158.302
C07881=1032.323,194.451,-108.538,169.725,43.882,158.302
C07882=1032.316,194.202,-108.514,169.721,43.884,158.302
C07883=1032.311,193.954,-108.490,169.719,43.885,158.302
C07884=1032.304,193.705,-108.466,169.715,43.886,158.302
C07885=1032.299,193.456,-108.442,169.712,43.888,158.302
C07886=1032.292,193.208,-108.417,169.708,43.889,158.302
C07887=1032.287,192.959,-108.393,169.705,43.890,158.302
C07888=1032.280,192.710,-108.369,169.701,43.892,158.302
C07889=1032.274,192.461,-108.344,169.699,43.893,158.302
C07890=1032.268,192.213,-108.321,169.695,43.894,158.302
C07891=1032.262,191.963,-108.296,169.692,43.895,158.302
C07892=1032.256,191.715,-108.272,169.688,43.896,158.302
C07893=1032.250,191.466,-108.248,169.685,43.898,158.302
C07894=1032.244,191.217,-108.224,169.681,43.899,158.301
C07895=1032.238,190.968,-108.199,169.678,43.900,158.301
C07896=1032.232,190.720,-108.176,169.675,43.902,158.301
C07897=1032.226,190.471,-108.151,169.672,43.903,158.301
C07898=1032.220,190.222,-108.127,169.668,43.904,158.301
C07899=1032.214,189.973,-108.103,169.665,43.906,158.301
C07900=1032.208,189.725,-108.079,169.661,43.907,158.301
C07901=1032.202,189.476,-108.055,169.658,43.908,158.301
C07902=1032.196,189.227,-108.031,169.656,43.909,158.301
C07903=1032.190,188.944,-108.003,169.652,43.911,158.301
C07904=1032.183,188.660,-107.976,169.648,43.912,158.301
C07905=1032.176,188.376,-107.949,169.644,43.914,158.301
C07906=1032.169,188.093,-107.921,169.640,43.915,158.301
C07907=1032.163,187.844,-107.897,169.637,43.916,158.301
C07908=1032.157,187.595,-107.873,169.634,43.918,158.301
C07909=1032.151,187.346,-107.848,169.631,43.919,158.301
C07910=1032.145,187.098,-107.825,169.627,43.920,158.301
C07911=1032.140,186.849,-107.801,169.624,43.922,158.301
C07912=1032.134,186.600,-107.777,169.620,43.923,158.301
C07913=1032.127,186.351,-107.754,169.618,43.924,158.301
C07914=1032.122,186.102,-107.729,169.615,43.925,158.301
C07915=1032.116,185.854,-107.705,169.611,43.927,158.301
C07916=1032.110,185.605,-107.681,169.608,43.928,158.301
C07917=1032.104,185.355,-107.658,169.604,43.930,158.301
C07918=1032.099,185.107,-107.633,169.601,43.931,158.301
C07919=1032.093,184.859,-107.610,169.599,43.932,158.301
C07920=1032.086,184.610,-107.586,169.595,43.933,158.301
C07921=1032.081,184.361,-107.562,169.592,43.935,158.301
C07922=1032.074,184.111,-107.538,169.588,43.936,158.301
C07923=1032.069,183.863,-107.514,169.585,43.937,158.301
C07924=1032.063,183.615,-107.490,169.583,43.938,158.301
C07925=1032.058,183.366,-107.466,169.579,43.940,158.301
C07926=1032.051,183.116,-107.443,169.576,43.941,158.301
C07927=1032.045,182.868,-107.419,169.573,43.942,158.301
C07928=1032.039,182.619,-107.396,169.569,43.944,158.301
C07929=1032.033,182.370,-107.372,169.566,43.945,158.301
C07930=1032.027,182.121,-107.349,169.563,43.947,158.301
C07931=1032.020,181.873,-107.326,169.560,43.948,158.301
C07932=1032.014,181.624,-107.303,169.556,43.950,158.301
C07933=1032.007,181.375,-107.279,169.554,43.952,158.301
C07934=1032.002,181.126,-107.256,169.550,43.953,158.301
C07935=1031.996,180.878,-107.232,169.547,43.954,158.301
C07936=1031.989,180.628,-107.209,169.544,43.956,158.301
C07937=1031.983,180.380,-107.185,169.541,43.958,158.301
C07938=1031.977,180.131,-107.163,169.538,43.959,158.301
C07939=1031.971,179.882,-107.140,169.534,43.961,158.301
C07940=1031.964,179.633,-107.116,169.531,43.962,158.301
C07941=1031.959,179.384,-107.093,169.528,43.963,158.301
C07942=1031.952,179.135,-107.069,169.525,43.965,158.301
C07943=1031.946,178.887,-107.046,169.522,43.967,158.301
C07944=1031.940,178.638,-107.024,169.518,43.968,158.301
C07945=1031.933,178.389,-107.000,169.516,43.970,158.302
C07946=1031.928,178.140,-106.977,169.513,43.971,158.302
C07947=1031.922,177.891,-106.954,169.509,43.973,158.301
C07948=1031.915,177.642,-106.930,169.506,43.974,158.302
C07949=1031.909,177.394,-106.907,169.503,43.976,158.302
C07950=1031.903,177.145,-106.884,169.500,43.977,158.302
C07951=1031.897,176.896,-106.861,169.497,43.979,158.302
C07952=1031.891,176.647,-106.837,169.493,43.980,158.302
C07953=1031.885,176.398,-106.814,169.491,43.982,158.302
C07954=1031.879,176.149,-106.791,169.488,43.983,158.302
C07955=1031.872,175.900,-106.768,169.484,43.985,158.302
C07956=1031.866,175.651,-106.745,169.481,43.986,158.302
C07957=1031.860,175.403,-106.722,169.478,43.988,158.302
C07958=1031.855,175.154,-106.699,169.475,43.989,158.302
C07959=1031.849,174.905,-106.676,169.472,43.991,158.302
C07960=1031.841,174.656,-106.653,169.468,43.993,158.302
C07961=1031.836,174.407,-106.630,169.466,43.994,158.302
C07962=1031.830,174.158,-106.607,169.463,43.996,158.302
C07963=1031.824,173.909,-106.584,169.459,43.997,158.302
C07964=1031.818,173.660,-106.560,169.456,43.999,158.302
C07965=1031.811,173.412,-106.538,169.454,44.000,158.302
C07966=1031.805,173.163,-106.515,169.450,44.002,158.302
C07967=1031.799,172.879,-106.489,169.447,44.004,158.302
C07968=1031.792,172.594,-106.462,169.444,44.005,158.302
C07969=1031.785,172.311,-106.436,169.440,44.007,158.302
C07970=1031.778,172.026,-106.410,169.436,44.009,158.302
C07971=1031.772,171.777,-106.387,169.434,44.011,158.303
C07972=1031.767,171.528,-106.364,169.431,44.012,158.303
C07973=1031.760,171.280,-106.341,169.427,44.014,158.303
C07974=1031.754,171.031,-106.318,169.424,44.015,158.303
C07975=1031.748,170.783,-106.295,169.422,44.016,158.303
C07976=1031.742,170.533,-106.272,169.419,44.018,158.303
C07977=1031.736,170.284,-106.249,169.415,44.020,158.303
C07978=1031.730,170.035,-106.226,169.413,44.021,158.303
C07979=1031.724,169.787,-106.204,169.410,44.023,158.303
C07980=1031.718,169.538,-106.181,169.407,44.024,158.303
C07981=1031.713,169.289,-106.158,169.403,44.026,158.303
C07982=1031.706,169.040,-106.135,169.400,44.027,158.303
C07983=1031.700,168.791,-106.112,169.398,44.029,158.303
C07984=1031.695,168.542,-106.089,169.394,44.031,158.303
C07985=1031.689,168.294,-106.066,169.391,44.032,158.303
C07986=1031.683,168.045,-106.043,169.389,44.034,158.303
C07987=1031.677,167.796,-106.021,169.386,44.035,158.303
C07988=1031.671,167.547,-105.998,169.383,44.036,158.303
C07989=1031.665,167.298,-105.975,169.379,44.038,158.303
C07990=1031.659,167.049,-105.952,169.377,44.039,158.303
C07991=1031.652,166.800,-105.930,169.374,44.041,158.303
C07992=1031.647,166.551,-105.907,169.371,44.043,158.303
C07993=1031.641,166.302,-105.884,169.367,44.044,158.303
C07994=1031.636,166.053,-105.861,169.365,44.046,158.304
C07995=1031.629,165.804,-105.839,169.362,44.047,158.304
C07996=1031.623,165.555,-105.816,169.359,44.049,158.304
C07997=1031.618,165.306,-105.793,169.357,44.050,158.304
C07998=1031.612,165.057,-105.770,169.353,44.052,158.304
C07999=1031.605,164.809,-105.748,169.350,44.054,158.304
C08000=1031.600,164.559,-105.726,169.347,44.055,158.304
C08001=1031.594,164.310,-105.703,169.345,44.057,158.304
C08002=1031.589,164.062,-105.680,169.342,44.058,158.304
C08003=1031.583,163.814,-105.658,169.338,44.060,158.304
C08004=1031.577,163.565,-105.635,169.335,44.061,158.304
C08005=1031.571,163.316,-105.612,169.333,44.063,158.304
C08006=1031.566,163.066,-105.590,169.330,44.064,158.304
C08007=1031.559,162.818,-105.567,169.327,44.066,158.304
C08008=1031.554,162.569,-105.544,169.324,44.068,158.304
C08009=1031.548,162.320,-105.521,169.321,44.069,158.304
C08010=1031.542,162.070,-105.499,169.318,44.070,158.304
C08011=1031.536,161.822,-105.477,169.315,44.072,158.304
C08012=1031.530,161.573,-105.454,169.313,44.073,158.304
C08013=1031.525,161.324,-105.431,169.310,44.075,158.305
C08014=1031.519,161.075,-105.409,169.306,44.077,158.305
C08015=1031.513,160.826,-105.386,169.304,44.079,158.305
C08016=1031.508,160.578,-105.364,169.301,44.080,158.305
C08017=1031.502,160.328,-105.342,169.298,44.081,158.305
C08018=1031.496,160.080,-105.319,169.295,44.083,158.305
C08019=1031.490,159.831,-105.296,169.293,44.084,158.305
C08020=1031.484,159.581,-105.274,169.290,44.086,158.305
C08021=1031.478,159.333,-105.252,169.286,44.087,158.305
C08022=1031.472,159.084,-105.230,169.284,44.089,158.305
C08023=1031.466,158.835,-105.207,169.281,44.091,158.305
C08024=1031.460,158.585,-105.185,169.278,44.093,158.305
C08025=1031.453,158.337,-105.163,169.276,44.094,158.305
C08026=1031.448,158.087,-105.141,169.272,44.096,158.306
C08027=1031.442,157.839,-105.119,169.269,44.098,158.306
C08028=1031.436,157.590,-105.097,169.267,44.100,158.306
C08029=1031.430,157.341,-105.074,169.264,44.101,158.306
C08030=1031.424,157.092,-105.053,169.261,44.103,158.306
C08031=1031.417,156.808,-105.027,169.258,44.105,158.306
C08032=1031.410,156.523,-105.003,169.254,44.107,158.306
C08033=1031.403,156.238,-104.977,169.251,44.109,158.306
C08034=1031.396,155.954,-104.951,169.248,44.111,158.306
C08035=1031.390,155.705,-104.930,169.245,44.112,158.306
C08036=1031.385,155.455,-104.907,169.242,44.114,158.306
C08037=1031.379,155.207,-104.885,169.240,44.116,158.307
C08038=1031.373,154.958,-104.864,169.236,44.117,158.306
C08039=1031.366,154.710,-104.841,169.233,44.119,158.307
C08040=1031.361,154.460,-104.819,169.231,44.121,158.307
C08041=1031.354,154.211,-104.798,169.228,44.122,158.307
C08042=1031.348,153.962,-104.775,169.225,44.124,158.307
C08043=1031.343,153.713,-104.753,169.223,44.126,158.307
C08044=1031.337,153.464,-104.732,169.220,44.127,158.307
C08045=1031.331,153.215,-104.710,169.216,44.130,158.307
C08046=1031.324,152.966,-104.688,169.214,44.131,158.307
C08047=1031.318,152.717,-104.666,169.211,44.133,158.307
C08048=1031.312,152.468,-104.644,169.208,44.135,158.307
C08049=1031.307,152.220,-104.623,169.206,44.136,158.308
C08050=1031.301,151.971,-104.600,169.203,44.138,158.308
C08051=1031.295,151.721,-104.579,169.199,44.140,158.308
C08052=1031.288,151.472,-104.557,169.197,44.142,158.308
C08053=1031.282,151.223,-104.535,169.194,44.144,158.308
C08054=1031.276,150.975,-104.513,169.191,44.145,158.308
C08055=1031.270,150.726,-104.492,169.189,44.147,158.308
C08056=1031.264,150.477,-104.470,169.186,44.149,158.308
C08057=1031.259,150.227,-104.448,169.184,44.151,158.308
C08058=1031.253,149.978,-104.426,169.181,44.152,158.308
C08059=1031.247,149.730,-104.405,169.177,44.154,158.308
C08060=1031.240,149.481,-104.383,169.175,44.156,158.309
C08061=1031.234,149.232,-104.361,169.172,44.157,158.309
C08062=1031.228,148.983,-104.339,169.169,44.159,158.309
C08063=1031.223,148.734,-104.318,169.167,44.161,158.309
C08064=1031.216,148.485,-104.296,169.164,44.163,158.309
C08065=1031.210,148.236,-104.275,169.161,44.164,158.309
C08066=1031.204,147.986,-104.253,169.159,44.166,158.309
C08067=1031.199,147.738,-104.232,169.156,44.168,158.309
C08068=1031.193,147.488,-104.210,169.153,44.170,158.309
C08069=1031.187,147.239,-104.188,169.150,44.171,158.309
C08070=1031.181,146.991,-104.167,169.147,44.173,158.310
C08071=1031.175,146.741,-104.145,169.145,44.175,158.310
C08072=1031.169,146.492,-104.124,169.142,44.177,158.310
C08073=1031.163,146.243,-104.102,169.139,44.179,158.310
C08074=1031.157,145.995,-104.081,169.137,44.180,158.310
C08075=1031.150,145.746,-104.060,169.134,44.182,158.310
C08076=1031.144,145.496,-104.038,169.131,44.184,158.310
C08077=1031.138,145.247,-104.016,169.128,44.186,158.310
C08078=1031.133,144.999,-103.995,169.125,44.188,158.311
C08079=1031.126,144.750,-103.973,169.123,44.190,158.311
C08080=1031.120,144.500,-103.952,169.120,44.192,158.311
C08081=1031.115,144.252,-103.930,169.117,44.193,158.311
C08082=1031.108,144.003,-103.909,169.115,44.195,158.311
C08083=1031.102,143.754,-103.888,169.112,44.197,158.311
C08084=1031.096,143.505,-103.867,169.109,44.199,158.311
C08085=1031.090,143.255,-103.846,169.107,44.200,158.311
C08086=1031.084,143.006,-103.824,169.103,44.203,158.311
C08087=1031.078,142.758,-103.803,169.100,44.204,158.311
C08088=1031.072,142.508,-103.781,169.098,44.206,158.312
C08089=1031.065,142.260,-103.760,169.095,44.208,158.312
C08090=1031.060,142.011,-103.739,169.093,44.210,158.312
C08091=1031.054,141.761,-103.718,169.090,44.211,158.312
C08092=1031.048,141.512,-103.696,169.088,44.213,158.312
C08093=1031.042,141.264,-103.675,169.085,44.215,158.312
C08094=1031.036,141.014,-103.653,169.082,44.216,158.312
C08095=1031.029,140.730,-103.629,169.079,44.219,158.312
C08096=1031.022,140.445,-103.606,169.076,44.220,158.313
C08097=1031.016,140.160,-103.581,169.073,44.223,158.313
C08098=1031.008,139.875,-103.556,169.070,44.225,158.313
C08099=1031.003,139.625,-103.535,169.067,44.226,158.313
C08100=1030.997,139.377,-103.514,169.065,44.228,158.313
C08101=1030.991,139.128,-103.492,169.062,44.230,158.313
C08102=1030.985,138.879,-103.472,169.059,44.232,158.313
C08103=1030.979,138.630,-103.451,169.057,44.234,158.314
C08104=1030.973,138.380,-103.429,169.054,44.236,158.314
C08105=1030.967,138.132,-103.408,169.051,44.238,158.314
C08106=1030.960,137.882,-103.388,169.048,44.240,158.314
C08107=1030.955,137.634,-103.366,169.045,44.242,158.314
C08108=1030.949,137.385,-103.345,169.043,44.243,158.314
C08109=1030.943,137.136,-103.325,169.040,44.245,158.314
C08110=1030.937,136.887,-103.303,169.038,44.247,158.314
C08111=1030.931,136.637,-103.282,169.035,44.249,158.314
C08112=1030.924,136.389,-103.262,169.032,44.251,158.315
C08113=1030.918,136.139,-103.240,169.030,44.253,158.315
C08114=1030.913,135.890,-103.219,169.027,44.255,158.315
C08115=1030.906,135.641,-103.198,169.025,44.256,158.315
C08116=1030.901,135.392,-103.178,169.022,44.258,158.315
C08117=1030.894,135.143,-103.157,169.019,44.260,158.315
C08118=1030.888,134.893,-103.136,169.017,44.262,158.315
C08119=1030.882,134.645,-103.115,169.014,44.264,158.316
C08120=1030.876,134.395,-103.094,169.012,44.266,158.316
C08121=1030.870,134.147,-103.073,169.009,44.268,158.316
C08122=1030.864,133.897,-103.053,169.006,44.269,158.316
C08123=1030.858,133.649,-103.031,169.004,44.271,158.316
C08124=1030.852,133.399,-103.011,169.001,44.273,158.316
C08125=1030.846,133.151,-102.990,168.998,44.275,158.316
C08126=1030.840,132.901,-102.969,168.995,44.277,158.316
C08127=1030.834,132.653,-102.948,168.992,44.279,158.317
C08128=1030.828,132.403,-102.927,168.990,44.281,158.317
C08129=1030.822,132.155,-102.907,168.987,44.283,158.317
C08130=1030.816,131.905,-102.886,168.985,44.285,158.317
C08131=1030.811,131.656,-102.865,168.982,44.287,158.317
C08132=1030.804,131.407,-102.844,168.979,44.289,158.317
C08133=1030.798,131.158,-102.824,168.977,44.290,158.317
C08134=1030.792,130.909,-102.802,168.974,44.292,158.318
C08135=1030.786,130.660,-102.782,168.972,44.294,158.318
C08136=1030.780,130.410,-102.762,168.969,44.296,158.318
C08137=1030.774,130.162,-102.740,168.967,44.298,158.318
C08138=1030.768,129.912,-102.720,168.964,44.300,158.318
C08139=1030.762,129.664,-102.700,168.961,44.302,158.318
C08140=1030.755,129.415,-102.679,168.959,44.304,158.318
C08141=1030.749,129.166,-102.658,168.956,44.306,158.318
C08142=1030.743,128.916,-102.638,168.954,44.308,158.319
C08143=1030.737,128.667,-102.618,168.951,44.310,158.319
C08144=1030.730,128.418,-102.598,168.948,44.311,158.319
C08145=1030.725,128.169,-102.577,168.946,44.313,158.319
C08146=1030.718,127.920,-102.556,168.943,44.315,158.319
C08147=1030.712,127.671,-102.536,168.941,44.318,158.319
C08148=1030.706,127.422,-102.516,168.938,44.320,158.320
C08149=1030.700,127.173,-102.495,168.936,44.322,158.320
C08150=1030.694,126.924,-102.475,168.933,44.324,158.320
C08151=1030.687,126.674,-102.454,168.931,44.326,158.320
C08152=1030.681,126.426,-102.434,168.928,44.327,158.320
C08153=1030.675,126.176,-102.414,168.925,44.329,158.320
C08154=1030.669,125.927,-102.394,168.923,44.331,158.320
C08155=1030.663,125.679,-102.373,168.920,44.333,158.321
C08156=1030.657,125.429,-102.353,168.917,44.335,158.321
C08157=1030.651,125.180,-102.332,168.914,44.337,158.321
C08158=1030.645,124.931,-102.312,168.912,44.339,158.321
C08159=1030.638,124.646,-102.289,168.909,44.342,158.321
C08160=1030.631,124.361,-102.265,168.907,44.344,158.321
C08161=1030.624,124.076,-102.242,168.903,44.346,158.321
C08162=1030.617,123.791,-102.218,168.901,44.348,158.322
C08163=1030.611,123.542,-102.198,168.898,44.350,158.322
C08164=1030.605,123.293,-102.178,168.895,44.352,158.322
C08165=1030.599,123.044,-102.158,168.893,44.354,158.322
C08166=1030.592,122.794,-102.138,168.890,44.356,158.322
C08167=1030.587,122.545,-102.117,168.888,44.358,158.322
C08168=1030.581,122.296,-102.097,168.885,44.360,158.323
C08169=1030.574,122.047,-102.077,168.883,44.362,158.323
C08170=1030.568,121.798,-102.057,168.880,44.364,158.323
C08171=1030.563,121.549,-102.036,168.877,44.366,158.323
C08172=1030.556,121.299,-102.016,168.875,44.368,158.323
C08173=1030.550,121.050,-101.996,168.872,44.370,158.323
C08174=1030.544,120.802,-101.976,168.870,44.371,158.323
C08175=1030.538,120.552,-101.956,168.867,44.373,158.324
C08176=1030.532,120.303,-101.935,168.864,44.375,158.324
C08177=1030.526,120.054,-101.915,168.862,44.377,158.324
C08178=1030.520,119.805,-101.895,168.860,44.380,158.324
C08179=1030.514,119.556,-101.875,168.857,44.382,158.324
C08180=1030.509,119.307,-101.855,168.854,44.384,158.324
C08181=1030.503,119.058,-101.835,168.852,44.386,158.325
C08182=1030.496,118.808,-101.814,168.849,44.387,158.325
C08183=1030.490,118.560,-101.794,168.847,44.389,158.325
C08184=1030.484,118.311,-101.774,168.844,44.391,158.325
C08185=1030.478,118.061,-101.753,168.842,44.393,158.325
C08186=1030.472,117.812,-101.733,168.839,44.395,158.325
C08187=1030.466,117.563,-101.714,168.836,44.397,158.325
C08188=1030.460,117.315,-101.694,168.835,44.399,158.326
C08189=1030.454,117.064,-101.674,168.832,44.401,158.326
C08190=1030.449,116.815,-101.653,168.830,44.403,158.326
C08191=1030.443,116.566,-101.633,168.827,44.405,158.326
C08192=1030.437,116.318,-101.613,168.824,44.407,158.326
C08193=1030.430,116.068,-101.593,168.822,44.408,158.326
C08194=1030.424,115.819,-101.573,168.819,44.410,158.326
C08195=1030.419,115.570,-101.553,168.817,44.412,158.326
C08196=1030.413,115.321,-101.533,168.814,44.414,158.327
C08197=1030.407,115.072,-101.513,168.812,44.416,158.327
C08198=1030.401,114.822,-101.493,168.809,44.418,158.327
C08199=1030.395,114.574,-101.473,168.806,44.420,158.327
C08200=1030.389,114.325,-101.453,168.804,44.422,158.327
C08201=1030.383,114.076,-101.433,168.802,44.424,158.327
C08202=1030.378,113.826,-101.413,168.800,44.426,158.328
C08203=1030.371,113.577,-101.393,168.797,44.427,158.328
C08204=1030.365,113.328,-101.373,168.795,44.429,158.328
C08205=1030.360,113.079,-101.353,168.792,44.431,158.328
C08206=1030.354,112.829,-101.333,168.789,44.433,158.328
C08207=1030.347,112.580,-101.313,168.787,44.435,158.328
C08208=1030.341,112.331,-101.293,168.784,44.437,158.328
C08209=1030.335,112.082,-101.274,168.782,44.439,158.328
C08210=1030.329,111.833,-101.254,168.779,44.441,158.329
C08211=1030.323,111.584,-101.234,168.776,44.443,158.329
C08212=1030.317,111.334,-101.215,168.774,44.445,158.329
C08213=1030.311,111.085,-101.195,168.772,44.447,158.329
C08214=1030.305,110.837,-101.175,168.769,44.449,158.329
C08215=1030.299,110.587,-101.156,168.767,44.451,158.329
C08216=1030.293,110.338,-101.136,168.765,44.453,158.330
C08217=1030.287,110.088,-101.116,168.762,44.455,158.330
C08218=1030.281,109.839,-101.096,168.760,44.457,158.330
C08219=1030.274,109.591,-101.077,168.757,44.459,158.330
C08220=1030.268,109.341,-101.058,168.755,44.461,158.330
C08221=1030.262,109.093,-101.038,168.752,44.463,158.330
C08222=1030.256,108.842,-101.018,168.750,44.465,158.331
C08223=1030.249,108.557,-100.996,168.746,44.467,158.331
C08224=1030.242,108.273,-100.973,168.744,44.470,158.331
C08225=1030.235,107.987,-100.951,168.741,44.472,158.331
C08226=1030.228,107.702,-100.929,168.738,44.475,158.331
C08227=1030.222,107.453,-100.910,168.735,44.477,158.331
C08228=1030.216,107.204,-100.890,168.733,44.479,158.332
C08229=1030.210,106.955,-100.871,168.730,44.481,158.332
C08230=1030.203,106.706,-100.851,168.729,44.483,158.332
C08231=1030.197,106.456,-100.832,168.726,44.485,158.332
C08232=1030.191,106.207,-100.812,168.723,44.487,158.332
C08233=1030.185,105.958,-100.793,168.721,44.489,158.332
C08234=1030.179,105.709,-100.773,168.718,44.491,158.333
C08235=1030.173,105.460,-100.754,168.716,44.493,158.333
C08236=1030.167,105.211,-100.735,168.713,44.495,158.333
C08237=1030.161,104.962,-100.715,168.711,44.497,158.333
C08238=1030.155,104.713,-100.696,168.708,44.499,158.333
C08239=1030.149,104.463,-100.676,168.706,44.501,158.333
C08240=1030.142,104.214,-100.657,168.703,44.503,158.334
C08241=1030.137,103.964,-100.638,168.701,44.505,158.334
C08242=1030.131,103.716,-100.618,168.698,44.507,158.334
C08243=1030.125,103.466,-100.599,168.696,44.509,158.334
C08244=1030.118,103.217,-100.580,168.694,44.511,158.334
C08245=1030.112,102.968,-100.560,168.691,44.513,158.334
C08246=1030.107,102.719,-100.541,168.689,44.515,158.335
C08247=1030.100,102.470,-100.521,168.686,44.517,158.335
C08248=1030.094,102.221,-100.502,168.684,44.519,158.335
C08249=1030.089,101.972,-100.483,168.681,44.521,158.335
C08250=1030.083,101.722,-100.464,168.679,44.523,158.335
C08251=1030.076,101.474,-100.444,168.676,44.525,158.335
C08252=1030.071,101.224,-100.425,168.674,44.527,158.335
C08253=1030.065,100.975,-100.406,168.671,44.529,158.336
C08254=1030.058,100.726,-100.386,168.670,44.531,158.336
C08255=1030.052,100.476,-100.367,168.667,44.533,158.336
C08256=1030.046,100.227,-100.347,168.664,44.535,158.336
C08257=1030.040,99.977,-100.328,168.662,44.537,158.336
C08258=1030.034,99.729,-100.309,168.659,44.539,158.336
C08259=1030.028,99.479,-100.290,168.657,44.541,158.337
C08260=1030.022,99.230,-100.271,168.654,44.543,158.337
C08261=1030.016,98.981,-100.252,168.652,44.545,158.337
C08262=1030.009,98.732,-100.233,168.649,44.548,158.337
C08263=1030.003,98.482,-100.214,168.647,44.550,158.337
C08264=1029.997,98.234,-100.194,168.644,44.552,158.337
C08265=1029.991,97.985,-100.176,168.642,44.554,158.338
C08266=1029.985,97.735,-100.157,168.640,44.556,158.338
C08267=1029.979,97.486,-100.138,168.638,44.558,158.338
C08268=1029.973,97.237,-100.119,168.635,44.560,158.338
C08269=1029.966,96.987,-100.100,168.633,44.562,158.338
C08270=1029.961,96.738,-100.081,168.630,44.564,158.339
C08271=1029.954,96.489,-100.062,168.628,44.566,158.339
C08272=1029.948,96.240,-100.044,168.625,44.568,158.339
C08273=1029.942,95.990,-100.024,168.623,44.570,158.339
C08274=1029.935,95.742,-100.005,168.620,44.572,158.339
C08275=1029.930,95.492,-99.986,168.618,44.575,158.339
C08276=1029.923,95.243,-99.967,168.615,44.577,158.339
C08277=1029.918,94.994,-99.948,168.612,44.579,158.340
C08278=1029.911,94.745,-99.929,168.610,44.581,158.340
C08279=1029.905,94.496,-99.910,168.609,44.583,158.340
C08280=1029.899,94.246,-99.891,168.606,44.585,158.340
C08281=1029.893,93.997,-99.873,168.603,44.587,158.340
C08282=1029.887,93.748,-99.853,168.601,44.589,158.340
C08283=1029.881,93.498,-99.835,168.598,44.591,158.341
C08284=1029.875,93.249,-99.815,168.596,44.593,158.341
C08285=1029.868,93.000,-99.797,168.593,44.595,158.341
C08286=1029.862,92.751,-99.778,168.591,44.597,158.341
C08287=1029.855,92.465,-99.757,168.588,44.599,158.341
C08288=1029.849,92.180,-99.735,168.586,44.602,158.342
C08289=1029.842,91.895,-99.713,168.582,44.604,158.342
C08290=1029.835,91.610,-99.692,168.580,44.607,158.342
C08291=1029.829,91.360,-99.673,168.577,44.609,158.342
C08292=1029.823,91.112,-99.655,168.575,44.610,158.342
C08293=1029.817,90.863,-99.636,168.572,44.612,158.342
C08294=1029.811,90.614,-99.617,168.571,44.615,158.343
C08295=1029.804,90.364,-99.598,168.568,44.617,158.343
C08296=1029.799,90.115,-99.579,168.566,44.619,158.343
C08297=1029.792,89.866,-99.560,168.563,44.621,158.343
C08298=1029.787,89.616,-99.541,168.561,44.623,158.343
C08299=1029.781,89.367,-99.523,168.558,44.625,158.343
C08300=1029.774,89.118,-99.504,168.556,44.627,158.344
C08301=1029.768,88.868,-99.486,168.553,44.629,158.344
C08302=1029.761,88.619,-99.467,168.550,44.631,158.344
C08303=1029.756,88.370,-99.450,168.548,44.634,158.344
C08304=1029.749,88.121,-99.431,168.546,44.636,158.344
C08305=1029.744,87.872,-99.412,168.544,44.637,158.344
C08306=1029.737,87.623,-99.393,168.542,44.640,158.345
C08307=1029.731,87.373,-99.374,168.539,44.642,158.345
C08308=1029.725,87.124,-99.357,168.537,44.644,158.345
C08309=1029.718,86.875,-99.338,168.534,44.646,158.345
C08310=1029.712,86.625,-99.319,168.532,44.648,158.345
C08311=1029.706,86.376,-99.301,168.529,44.650,158.345
C08312=1029.700,86.127,-99.283,168.526,44.652,158.346
C08313=1029.693,85.878,-99.264,168.524,44.655,158.346
C08314=1029.688,85.629,-99.245,168.522,44.657,158.346
C08315=1029.682,85.379,-99.227,168.519,44.659,158.346
C08316=1029.675,85.130,-99.209,168.518,44.661,158.346
C08317=1029.669,84.881,-99.190,168.515,44.663,158.347
C08318=1029.663,84.632,-99.172,168.513,44.665,158.347
C08319=1029.657,84.383,-99.154,168.510,44.667,158.347
C08320=1029.650,84.133,-99.135,168.508,44.670,158.347
C08321=1029.644,83.884,-99.117,168.505,44.672,158.347
C08322=1029.638,83.635,-99.098,168.502,44.674,158.347
C08323=1029.632,83.385,-99.079,168.500,44.676,158.348
C08324=1029.627,83.136,-99.062,168.498,44.678,158.348
C08325=1029.620,82.887,-99.043,168.495,44.680,158.348
C08326=1029.614,82.637,-99.025,168.493,44.682,158.348
C08327=1029.608,82.388,-99.006,168.491,44.684,158.348
C08328=1029.601,82.139,-98.988,168.489,44.686,158.349
C08329=1029.596,81.890,-98.970,168.486,44.688,158.349
C08330=1029.589,81.641,-98.952,168.483,44.690,158.349
C08331=1029.583,81.391,-98.934,168.481,44.692,158.349
C08332=1029.577,81.142,-98.915,168.478,44.694,158.349
C08333=1029.572,80.893,-98.896,168.476,44.697,158.349
C08334=1029.566,80.644,-98.878,168.473,44.699,158.349
C08335=1029.559,80.394,-98.859,168.472,44.701,158.350
C08336=1029.553,80.145,-98.842,168.469,44.703,158.350
C08337=1029.547,79.896,-98.823,168.467,44.705,158.350
C08338=1029.541,79.647,-98.805,168.464,44.707,158.350
C08339=1029.535,79.397,-98.787,168.462,44.709,158.350
C08340=1029.529,79.148,-98.769,168.459,44.711,158.350
C08341=1029.523,78.899,-98.750,168.457,44.713,158.351
C08342=1029.517,78.649,-98.733,168.455,44.715,158.351
C08343=1029.510,78.400,-98.714,168.453,44.717,158.351
C08344=1029.505,78.150,-98.695,168.450,44.719,158.351
C08345=1029.499,77.902,-98.677,168.448,44.721,158.351
C08346=1029.493,77.652,-98.659,168.445,44.723,158.351
C08347=1029.486,77.403,-98.641,168.443,44.726,158.352
C08348=1029.480,77.154,-98.623,168.440,44.728,158.352
C08349=1029.474,76.905,-98.606,168.437,44.730,158.352
C08350=1029.468,76.655,-98.587,168.435,44.732,158.352
C08351=1029.460,76.370,-98.566,168.433,44.734,158.352
C08352=1029.453,76.085,-98.546,168.430,44.737,158.353
C08353=1029.447,75.799,-98.524,168.428,44.739,158.353
C08354=1029.440,75.514,-98.505,168.424,44.742,158.353
C08355=1029.433,75.265,-98.487,168.422,44.744,158.353
C08356=1029.427,75.015,-98.469,168.419,44.746,158.353
C08357=1029.421,74.766,-98.451,168.417,44.748,158.353
C08358=1029.415,74.517,-98.433,168.415,44.750,158.354
C08359=1029.409,74.268,-98.415,168.413,44.752,158.354
C08360=1029.403,74.018,-98.397,168.410,44.755,158.354
C08361=1029.396,73.770,-98.379,168.408,44.757,158.354
C08362=1029.390,73.520,-98.361,168.405,44.758,158.354
C08363=1029.384,73.270,-98.343,168.403,44.761,158.355
C08364=1029.378,73.021,-98.326,168.400,44.763,158.355
C08365=1029.372,72.772,-98.307,168.398,44.765,158.355
C08366=1029.365,72.523,-98.290,168.395,44.767,158.355
C08367=1029.360,72.274,-98.272,168.394,44.769,158.355
C08368=1029.353,72.024,-98.253,168.391,44.771,158.355
C08369=1029.347,71.775,-98.235,168.389,44.773,158.356
C08370=1029.342,71.526,-98.218,168.386,44.775,158.356
C08371=1029.335,71.276,-98.201,168.384,44.778,158.356
C08372=1029.329,71.027,-98.183,168.381,44.780,158.356
C08373=1029.323,70.778,-98.164,168.379,44.782,158.356
C08374=1029.317,70.528,-98.146,168.376,44.784,158.356
C08375=1029.310,70.280,-98.129,168.374,44.786,158.357
C08376=1029.304,70.030,-98.111,168.372,44.788,158.357
C08377=1029.298,69.780,-98.094,168.370,44.790,158.357
C08378=1029.293,69.531,-98.076,168.367,44.793,158.357
C08379=1029.285,69.282,-98.058,168.365,44.795,158.357
C08380=1029.280,69.033,-98.040,168.362,44.797,158.357
C08381=1029.274,68.783,-98.022,168.360,44.799,158.358
C08382=1029.268,68.534,-98.004,168.357,44.801,158.358
C08383=1029.261,68.285,-97.988,168.355,44.803,158.358
C08384=1029.255,68.035,-97.970,168.352,44.805,158.358
C08385=1029.248,67.786,-97.952,168.351,44.808,158.358
C08386=1029.243,67.537,-97.935,168.348,44.810,158.358
C08387=1029.237,67.287,-97.917,168.346,44.812,158.359
C08388=1029.231,67.038,-97.900,168.343,44.814,158.359
C08389=1029.224,66.789,-97.882,168.341,44.816,158.359
C08390=1029.219,66.540,-97.864,168.338,44.818,158.359
C08391=1029.212,66.291,-97.846,168.336,44.820,158.359
C08392=1029.206,66.041,-97.828,168.333,44.823,158.360
C08393=1029.199,65.792,-97.811,168.331,44.825,158.360
C08394=1029.193,65.543,-97.793,168.328,44.827,158.360
C08395=1029.188,65.294,-97.776,168.327,44.829,158.360
C08396=1029.181,65.044,-97.758,168.324,44.831,158.360
C08397=1029.175,64.794,-97.741,168.322,44.833,158.360
C08398=1029.168,64.546,-97.724,168.319,44.835,158.360
C08399=1029.162,64.296,-97.706,168.317,44.838,158.361
C08400=1029.156,64.047,-97.689,168.314,44.840,158.361
C08401=1029.150,63.797,-97.671,168.312,44.842,158.361
C08402=1029.144,63.548,-97.654,168.309,44.844,158.361
C08403=1029.138,63.298,-97.637,168.307,44.846,158.361
C08404=1029.132,63.050,-97.620,168.304,44.848,158.361
C08405=1029.126,62.800,-97.602,168.302,44.851,158.362
C08406=1029.119,62.550,-97.584,168.299,44.853,158.362
C08407=1029.112,62.302,-97.567,168.297,44.855,158.362
C08408=1029.106,62.052,-97.551,168.295,44.857,158.362
C08409=1029.100,61.803,-97.533,168.293,44.860,158.363
C08410=1029.093,61.553,-97.516,168.291,44.862,158.363
C08411=1029.087,61.304,-97.499,168.288,44.864,158.363
C08412=1029.080,61.055,-97.481,168.286,44.866,158.363
C08413=1029.075,60.805,-97.465,168.283,44.868,158.363
C08414=1029.068,60.556,-97.447,168.281,44.871,158.364
C08415=1029.062,60.310,-97.431,168.278,44.873,158.364
C08416=1029.056,60.063,-97.413,168.276,44.876,158.364
C08417=1029.050,59.816,-97.397,168.273,44.878,158.364
C08418=1029.043,59.569,-97.380,168.271,44.879,158.364
C08419=1029.037,59.323,-97.362,168.268,44.882,158.364
C08420=1029.031,59.076,-97.345,168.266,44.884,158.365
C08421=1029.025,58.830,-97.329,168.263,44.886,158.365
C08422=1029.019,58.584,-97.311,168.262,44.889,158.365
C08423=1029.012,58.334,-97.295,168.259,44.890,158.365
C08424=1029.006,58.085,-97.278,168.257,44.893,158.365
C08425=1029.000,57.835,-97.260,168.254,44.895,158.366
C08426=1028.994,57.587,-97.243,168.252,44.897,158.366
C08427=1028.987,57.337,-97.226,168.250,44.900,158.366
C08428=1028.981,57.088,-97.209,168.247,44.902,158.366
C08429=1028.975,56.838,-97.191,168.244,44.904,158.366
C08430=1028.969,56.589,-97.175,168.242,44.906,158.366
C08431=1028.962,56.339,-97.158,168.239,44.908,158.367
C08432=1028.956,56.091,-97.141,168.237,44.910,158.367
C08433=1028.950,55.840,-97.124,168.235,44.913,158.367
C08434=1028.944,55.591,-97.107,168.232,44.915,158.367
C08435=1028.938,55.342,-97.090,168.230,44.917,158.367
C08436=1028.931,55.093,-97.073,168.227,44.919,158.367
C08437=1028.925,54.844,-97.055,168.226,44.921,158.368
C08438=1028.919,54.594,-97.039,168.223,44.924,158.368
C08439=1028.912,54.303,-97.019,168.220,44.926,158.368
C08440=1028.904,54.012,-96.999,168.217,44.929,158.368
C08441=1028.897,53.721,-96.979,168.214,44.932,158.368
C08442=1028.889,53.430,-96.959,168.211,44.934,158.369
C08443=1028.883,53.181,-96.943,168.209,44.936,158.369
C08444=1028.878,52.932,-96.925,168.207,44.938,158.369
C08445=1028.871,52.682,-96.909,168.204,44.940,158.369
C08446=1028.865,52.433,-96.892,168.202,44.943,158.369
C08447=1028.859,52.184,-96.875,168.199,44.945,158.369
C08448=1028.853,51.934,-96.858,168.198,44.947,158.370
C08449=1028.847,51.685,-96.841,168.195,44.949,158.370
C08450=1028.840,51.435,-96.824,168.193,44.951,158.370
C08451=1028.834,51.186,-96.807,168.190,44.953,158.370
C08452=1028.829,50.937,-96.790,168.188,44.955,158.370
C08453=1028.822,50.687,-96.773,168.185,44.958,158.371
C08454=1028.816,50.438,-96.757,168.183,44.960,158.371
C08455=1028.810,50.189,-96.740,168.180,44.962,158.371
C08456=1028.803,49.939,-96.723,168.177,44.964,158.371
C08457=1028.798,49.690,-96.705,168.175,44.966,158.371
C08458=1028.792,49.441,-96.689,168.173,44.968,158.371
C08459=1028.785,49.191,-96.672,168.171,44.970,158.371
C08460=1028.779,48.942,-96.656,168.169,44.973,158.372
C08461=1028.774,48.692,-96.639,168.166,44.975,158.372
C08462=1028.767,48.443,-96.621,168.164,44.977,158.372
C08463=1028.761,48.194,-96.605,168.161,44.979,158.372
C08464=1028.755,47.945,-96.588,168.158,44.981,158.372
C08465=1028.749,47.695,-96.572,168.156,44.983,158.372
C08466=1028.742,47.446,-96.554,168.154,44.985,158.373
C08467=1028.737,47.196,-96.538,168.151,44.987,158.373
C08468=1028.731,46.947,-96.521,168.149,44.989,158.373
C08469=1028.724,46.698,-96.504,168.147,44.992,158.373
C08470=1028.718,46.448,-96.487,168.145,44.994,158.373
C08471=1028.712,46.199,-96.470,168.142,44.996,158.373
C08472=1028.706,45.950,-96.454,168.139,44.998,158.373
C08473=1028.700,45.700,-96.437,168.137,45.000,158.374
C08474=1028.693,45.451,-96.420,168.135,45.002,158.374
C08475=1028.688,45.201,-96.404,168.132,45.004,158.374
C08476=1028.682,44.952,-96.387,168.129,45.006,158.374
C08477=1028.675,44.703,-96.370,168.128,45.008,158.374
C08478=1028.669,44.453,-96.354,168.125,45.010,158.374
C08479=1028.663,44.168,-96.334,168.122,45.013,158.375
C08480=1028.656,43.882,-96.315,168.119,45.015,158.375
C08481=1028.649,43.597,-96.296,168.117,45.017,158.375
C08482=1028.642,43.310,-96.277,168.113,45.020,158.375
C08483=1028.636,43.061,-96.261,168.112,45.022,158.375
C08484=1028.630,42.812,-96.243,168.110,45.024,158.375
C08485=1028.623,42.562,-96.227,168.107,45.026,158.376
C08486=1028.617,42.313,-96.211,168.104,45.028,158.376
C08487=1028.611,42.064,-96.195,168.102,45.031,158.376
C08488=1028.605,41.814,-96.179,168.100,45.033,158.376
C08489=1028.598,41.565,-96.161,168.097,45.035,158.376
C08490=1028.593,41.315,-96.145,168.095,45.037,158.376
C08491=1028.587,41.066,-96.129,168.092,45.039,158.377
C08492=1028.581,40.817,-96.112,168.090,45.041,158.377
C08493=1028.575,40.567,-96.096,168.087,45.044,158.377
C08494=1028.568,40.317,-96.080,168.085,45.046,158.377
C08495=1028.562,40.069,-96.063,168.082,45.048,158.377
C08496=1028.556,39.819,-96.046,168.080,45.050,158.377
C08497=1028.550,39.570,-96.030,168.078,45.052,158.378
C08498=1028.544,39.321,-96.014,168.076,45.054,158.378
C08499=1028.537,39.071,-95.998,168.073,45.056,158.378
C08500=1028.531,38.821,-95.982,168.071,45.059,158.378
C08501=1028.525,38.572,-95.965,168.068,45.061,158.378
C08502=1028.519,38.323,-95.949,168.066,45.063,158.378
C08503=1028.513,38.073,-95.933,168.063,45.065,158.378
C08504=1028.507,37.824,-95.917,168.061,45.068,158.379
C08505=1028.500,37.575,-95.899,168.058,45.070,158.379
C08506=1028.494,37.325,-95.883,168.056,45.072,158.379
C08507=1028.488,37.076,-95.867,168.053,45.074,158.379
C08508=1028.482,36.827,-95.850,168.051,45.076,158.379
C08509=1028.476,36.578,-95.835,168.048,45.078,158.379
C08510=1028.470,36.328,-95.819,168.046,45.081,158.380
C08511=1028.463,36.078,-95.803,168.043,45.083,158.380
C08512=1028.457,35.828,-95.787,168.041,45.085,158.380
C08513=1028.451,35.579,-95.771,168.038,45.087,158.380
C08514=1028.445,35.330,-95.754,168.036,45.089,158.380
C08515=1028.438,35.081,-95.739,168.033,45.091,158.380
C08516=1028.432,34.831,-95.723,168.031,45.094,158.381
C08517=1028.426,34.581,-95.706,168.028,45.096,158.381
C08518=1028.420,34.332,-95.690,168.026,45.099,158.381
C08519=1028.413,34.083,-95.674,168.025,45.101,158.381
C08520=1028.407,33.834,-95.658,168.022,45.103,158.381
C08521=1028.401,33.584,-95.641,168.020,45.105,158.382
C08522=1028.395,33.335,-95.627,168.017,45.107,158.382
C08523=1028.389,33.085,-95.610,168.014,45.109,158.382
C08524=1028.383,32.836,-95.594,168.012,45.112,158.382
C08525=1028.376,32.587,-95.578,168.010,45.114,158.382
C08526=1028.370,32.337,-95.562,168.007,45.116,158.382
C08527=1028.364,32.087,-95.545,168.005,45.119,158.383
C08528=1028.357,31.838,-95.530,168.002,45.121,158.383
C08529=1028.351,31.588,-95.514,168.000,45.122,158.383
C08530=1028.345,31.339,-95.498,167.997,45.125,158.383
C08531=1028.339,31.090,-95.482,167.995,45.127,158.383
C08532=1028.333,30.841,-95.466,167.992,45.129,158.383
C08533=1028.327,30.591,-95.450,167.990,45.132,158.384
C08534=1028.320,30.342,-95.435,167.987,45.134,158.384
C08535=1028.314,30.092,-95.419,167.985,45.136,158.384
C08536=1028.308,29.843,-95.402,167.982,45.138,158.384
C08537=1028.302,29.594,-95.387,167.980,45.140,158.384
C08538=1028.296,29.345,-95.370,167.977,45.142,158.384
C08539=1028.290,29.095,-95.355,167.975,45.144,158.384
C08540=1028.283,28.846,-95.339,167.972,45.147,158.385
C08541=1028.277,28.596,-95.323,167.970,45.149,158.385
C08542=1028.272,28.346,-95.307,167.967,45.151,158.385
C08543=1028.264,28.060,-95.289,167.965,45.154,158.385
C08544=1028.257,27.775,-95.271,167.961,45.156,158.385
C08545=1028.250,27.489,-95.253,167.959,45.159,158.385
C08546=1028.243,27.203,-95.234,167.957,45.161,158.386
C08547=1028.236,26.953,-95.219,167.954,45.163,158.386
C08548=1028.230,26.704,-95.203,167.952,45.166,158.386
C08549=1028.224,26.455,-95.187,167.949,45.168,158.386
C08550=1028.217,26.205,-95.172,167.947,45.170,158.386
C08551=1028.211,25.956,-95.156,167.944,45.173,158.387
C08552=1028.205,25.706,-95.141,167.942,45.175,158.387
C08553=1028.199,25.457,-95.125,167.939,45.177,158.387
C08554=1028.192,25.208,-95.109,167.937,45.179,158.387
C08555=1028.187,24.958,-95.094,167.934,45.181,158.387
C08556=1028.180,24.709,-95.078,167.932,45.183,158.387
C08557=1028.174,24.459,-95.063,167.930,45.186,158.388
C08558=1028.168,24.210,-95.047,167.927,45.188,158.388
C08559=1028.161,23.960,-95.032,167.925,45.191,158.388
C08560=1028.155,23.711,-95.016,167.922,45.193,158.388
C08561=1028.150,23.462,-95.001,167.920,45.195,158.388
C08562=1028.144,23.213,-94.985,167.917,45.197,158.388
C08563=1028.137,22.963,-94.970,167.915,45.199,158.388
C08564=1028.131,22.714,-94.954,167.912,45.201,158.389
C08565=1028.125,22.464,-94.939,167.910,45.204,158.389
C08566=1028.118,22.215,-94.923,167.907,45.206,158.389
C08567=1028.113,21.965,-94.908,167.905,45.208,158.389
C08568=1028.106,21.716,-94.892,167.902,45.211,158.389
C08569=1028.100,21.466,-94.876,167.900,45.213,158.389
C08570=1028.094,21.217,-94.861,167.897,45.215,158.390
C08571=1028.087,20.967,-94.846,167.895,45.217,158.390
C08572=1028.081,20.718,-94.829,167.892,45.219,158.390
C08573=1028.075,20.468,-94.814,167.890,45.221,158.390
C08574=1028.069,20.219,-94.798,167.887,45.223,158.390
C08575=1028.062,19.969,-94.783,167.885,45.226,158.390
C08576=1028.057,19.720,-94.769,167.882,45.228,158.391
C08577=1028.051,19.471,-94.752,167.879,45.230,158.391
C08578=1028.044,19.221,-94.738,167.876,45.233,158.391
C08579=1028.038,18.972,-94.722,167.874,45.235,158.391
C08580=1028.032,18.722,-94.706,167.872,45.238,158.391
C08581=1028.026,18.473,-94.691,167.869,45.240,158.391
C08582=1028.019,18.224,-94.676,167.866,45.242,158.391
C08583=1028.013,17.974,-94.661,167.864,45.244,158.392
C08584=1028.007,17.724,-94.645,167.862,45.246,158.392
C08585=1028.001,17.476,-94.630,167.859,45.248,158.392
C08586=1027.994,17.226,-94.615,167.857,45.251,158.392
C08587=1027.989,16.976,-94.599,167.854,45.253,158.392
C08588=1027.982,16.726,-94.584,167.852,45.255,158.392
C08589=1027.976,16.477,-94.569,167.849,45.258,158.393
C08590=1027.969,16.228,-94.554,167.847,45.260,158.393
C08591=1027.964,15.978,-94.538,167.844,45.262,158.393
C08592=1027.958,15.729,-94.523,167.842,45.264,158.393
C08593=1027.951,15.480,-94.508,167.839,45.266,158.393
C08594=1027.945,15.230,-94.493,167.837,45.268,158.393
C08595=1027.939,14.980,-94.478,167.834,45.271,158.394
C08596=1027.933,14.731,-94.462,167.832,45.273,158.394
C08597=1027.926,14.481,-94.447,167.829,45.275,158.394
C08598=1027.920,14.232,-94.432,167.827,45.278,158.394
C08599=1027.915,13.983,-94.417,167.824,45.280,158.394
C08600=1027.908,13.733,-94.402,167.822,45.282,158.394
C08601=1027.902,13.483,-94.387,167.819,45.284,158.394
C08602=1027.895,13.234,-94.371,167.817,45.286,158.395
C08603=1027.889,12.984,-94.356,167.815,45.289,158.395
C08604=1027.883,12.736,-94.342,167.811,45.291,158.395
C08605=1027.877,12.486,-94.327,167.809,45.294,158.395
C08606=1027.870,12.236,-94.312,167.806,45.296,158.395
C08607=1027.863,11.952,-94.295,167.804,45.299,158.396
C08608=1027.856,11.668,-94.278,167.800,45.302,158.396
C08609=1027.849,11.383,-94.261,167.798,45.304,158.396
C08610=1027.841,11.098,-94.245,167.795,45.307,158.396
C08611=1027.835,10.849,-94.230,167.792,45.309,158.396
C08612=1027.829,10.599,-94.215,167.790,45.311,158.396
C08613=1027.823,10.350,-94.200,167.787,45.313,158.396
C08614=1027.816,10.101,-94.184,167.785,45.316,158.397
C08615=1027.810,9.851,-94.169,167.782,45.318,158.397
C08616=1027.803,9.602,-94.155,167.780,45.321,158.397
C08617=1027.798,9.353,-94.140,167.776,45.323,158.397
C08618=1027.791,9.103,-94.125,167.774,45.326,158.397
C08619=1027.785,8.853,-94.111,167.772,45.328,158.398
C08620=1027.779,8.603,-94.096,167.769,45.330,158.398
C08621=1027.773,8.354,-94.081,167.767,45.332,158.398
C08622=1027.767,8.104,-94.066,167.764,45.334,158.398
C08623=1027.760,7.855,-94.051,167.762,45.337,158.398
C08624=1027.754,7.605,-94.036,167.759,45.339,158.398
C08625=1027.748,7.356,-94.022,167.757,45.341,158.398
C08626=1027.742,7.107,-94.007,167.754,45.344,158.399
C08627=1027.735,6.857,-93.992,167.752,45.346,158.399
C08628=1027.729,6.607,-93.977,167.748,45.349,158.399
C08629=1027.723,6.358,-93.962,167.746,45.351,158.399
C08630=1027.717,6.109,-93.947,167.743,45.353,158.399
C08631=1027.710,5.859,-93.933,167.741,45.355,158.399
C08632=1027.705,5.610,-93.918,167.738,45.357,158.400
C08633=1027.698,5.360,-93.904,167.736,45.359,158.400
C08634=1027.691,5.110,-93.889,167.734,45.362,158.400
C08635=1027.686,4.861,-93.875,167.731,45.364,158.400
C08636=1027.679,4.612,-93.860,167.728,45.366,158.400
C08637=1027.673,4.362,-93.845,167.726,45.369,158.400
C08638=1027.667,4.113,-93.830,167.724,45.371,158.400
C08639=1027.661,3.863,-93.815,167.721,45.373,158.401
C08640=1027.655,3.613,-93.801,167.718,45.376,158.401
C08641=1027.649,3.364,-93.787,167.715,45.378,158.401
C08642=1027.642,3.115,-93.772,167.713,45.380,158.401
C08643=1027.637,2.866,-93.757,167.710,45.382,158.401
C08644=1027.630,2.616,-93.742,167.708,45.384,158.401
C08645=1027.624,2.366,-93.728,167.705,45.386,158.401
C08646=1027.618,2.117,-93.713,167.703,45.389,158.402
C08647=1027.612,1.867,-93.698,167.700,45.391,158.402
C08648=1027.606,1.617,-93.683,167.698,45.393,158.402
C08649=1027.600,1.368,-93.669,167.695,45.396,158.402
C08650=1027.593,1.119,-93.655,167.693,45.398,158.402
C08651=1027.587,0.870,-93.641,167.690,45.400,158.402
C08652=1027.581,0.620,-93.626,167.687,45.403,158.403
C08653=1027.574,0.370,-93.611,167.684,45.405,158.403
C08654=1027.569,0.121,-93.597,167.682,45.407,158.403
C08655=1027.563,-0.129,-93.582,167.679,45.409,158.403
C08656=1027.557,-0.378,-93.567,167.677,45.412,158.403
C08657=1027.551,-0.628,-93.553,167.674,45.414,158.403
C08658=1027.545,-0.877,-93.538,167.672,45.416,158.403
C08659=1027.539,-1.127,-93.524,167.669,45.418,158.403
C08660=1027.533,-1.376,-93.509,167.667,45.420,158.404
C08661=1027.527,-1.626,-93.495,167.664,45.422,158.404
C08662=1027.521,-1.875,-93.480,167.662,45.424,158.404
C08663=1027.514,-2.124,-93.466,167.660,45.427,158.404
C08664=1027.508,-2.375,-93.452,167.656,45.429,158.404
C08665=1027.502,-2.624,-93.437,167.653,45.431,158.404
C08666=1027.496,-2.874,-93.423,167.651,45.433,158.404
C08667=1027.490,-3.123,-93.408,167.648,45.435,158.404
C08668=1027.484,-3.372,-93.393,167.646,45.438,158.405
C08669=1027.478,-3.622,-93.379,167.643,45.440,158.405
C08670=1027.472,-3.872,-93.364,167.641,45.442,158.405
C08671=1027.465,-4.154,-93.349,167.638,45.445,158.405
C08672=1027.458,-4.436,-93.332,167.635,45.448,158.405
C08673=1027.451,-4.719,-93.317,167.632,45.450,158.405
C08674=1027.444,-5.002,-93.301,167.629,45.453,158.406
C08675=1027.437,-5.251,-93.287,167.626,45.456,158.406
C08676=1027.432,-5.500,-93.273,167.624,45.458,158.406
C08677=1027.425,-5.750,-93.258,167.621,45.460,158.406
C08678=1027.419,-5.999,-93.245,167.619,45.462,158.406
C08679=1027.413,-6.249,-93.230,167.616,45.464,158.406
C08680=1027.406,-6.498,-93.216,167.614,45.467,158.407
C08681=1027.400,-6.749,-93.202,167.610,45.469,158.407
C08682=1027.394,-6.997,-93.188,167.608,45.472,158.407
C08683=1027.388,-7.247,-93.174,167.605,45.474,158.407
C08684=1027.382,-7.496,-93.159,167.603,45.477,158.407
C08685=1027.375,-7.746,-93.146,167.600,45.479,158.407
C08686=1027.370,-7.996,-93.132,167.598,45.481,158.407
C08687=1027.363,-8.245,-93.117,167.595,45.484,158.408
C08688=1027.357,-8.495,-93.104,167.592,45.486,158.408
C08689=1027.350,-8.744,-93.089,167.590,45.488,158.408
C08690=1027.344,-8.994,-93.075,167.587,45.490,158.408
C08691=1027.338,-9.244,-93.062,167.585,45.492,158.408
C08692=1027.332,-9.493,-93.047,167.581,45.495,158.408
C08693=1027.326,-9.742,-93.033,167.579,45.497,158.408
C08694=1027.320,-9.992,-93.020,167.576,45.500,158.409
C08695=1027.314,-10.241,-93.005,167.574,45.502,158.409
C08696=1027.307,-10.491,-92.991,167.571,45.504,158.409
C08697=1027.301,-10.741,-92.978,167.569,45.507,158.409
C08698=1027.295,-10.991,-92.964,167.565,45.509,158.409
C08699=1027.289,-11.240,-92.949,167.563,45.511,158.409
C08700=1027.283,-11.489,-92.936,167.561,45.514,158.410
C08701=1027.277,-11.739,-92.922,167.558,45.516,158.410
C08702=1027.270,-11.988,-92.908,167.555,45.518,158.410
C08703=1027.265,-12.237,-92.894,167.553,45.521,158.410
C08704=1027.259,-12.488,-92.880,167.550,45.523,158.410
C08705=1027.252,-12.737,-92.866,167.547,45.526,158.410
C08706=1027.246,-12.987,-92.852,167.545,45.528,158.410
C08707=1027.240,-13.236,-92.838,167.542,45.530,158.410
C08708=1027.234,-13.485,-92.824,167.540,45.532,158.411
C08709=1027.227,-13.735,-92.811,167.537,45.534,158.411
C08710=1027.222,-13.985,-92.797,167.534,45.537,158.411
C08711=1027.215,-14.234,-92.783,167.531,45.539,158.411
C08712=1027.209,-14.484,-92.769,167.529,45.541,158.411
C08713=1027.203,-14.733,-92.755,167.526,45.543,158.411
C08714=1027.198,-14.983,-92.742,167.524,45.545,158.411
C08715=1027.191,-15.233,-92.728,167.521,45.548,158.412
C08716=1027.185,-15.482,-92.714,167.518,45.550,158.412
C08717=1027.179,-15.732,-92.701,167.515,45.552,158.412
C08718=1027.173,-15.982,-92.687,167.513,45.555,158.412
C08719=1027.167,-16.231,-92.673,167.510,45.557,158.412
C08720=1027.160,-16.480,-92.659,167.507,45.560,158.412
C08721=1027.154,-16.730,-92.646,167.505,45.562,158.412
C08722=1027.148,-16.979,-92.632,167.502,45.565,158.413
C08723=1027.142,-17.229,-92.619,167.500,45.567,158.413
C08724=1027.135,-17.479,-92.605,167.496,45.570,158.413
C08725=1027.130,-17.728,-92.591,167.494,45.572,158.413
C08726=1027.123,-17.977,-92.578,167.492,45.574,158.413
C08727=1027.117,-18.227,-92.564,167.489,45.577,158.413
C08728=1027.110,-18.477,-92.551,167.487,45.579,158.414
C08729=1027.105,-18.726,-92.537,167.483,45.581,158.414
C08730=1027.099,-18.975,-92.524,167.481,45.584,158.414
C08731=1027.092,-19.226,-92.511,167.478,45.586,158.414
C08732=1027.086,-19.475,-92.498,167.476,45.588,158.414
C08733=1027.080,-19.725,-92.484,167.472,45.591,158.414
C08734=1027.074,-19.974,-92.470,167.470,45.593,158.414
C08735=1027.067,-20.255,-92.455,167.466,45.596,158.414
C08736=1027.060,-20.536,-92.440,167.464,45.599,158.415
C08737=1027.054,-20.817,-92.425,167.461,45.601,158.415
C08738=1027.046,-21.098,-92.410,167.457,45.604,158.415
C08739=1027.040,-21.347,-92.396,167.455,45.607,158.415
C08740=1027.034,-21.597,-92.383,167.452,45.609,158.415
C08741=1027.027,-21.847,-92.369,167.450,45.611,158.415
C08742=1027.021,-22.096,-92.356,167.448,45.614,158.416
C08743=1027.015,-22.346,-92.343,167.444,45.616,158.416
C08744=1027.010,-22.595,-92.329,167.442,45.619,158.416
C08745=1027.004,-22.845,-92.316,167.439,45.621,158.416
C08746=1026.997,-23.095,-92.302,167.437,45.623,158.416
C08747=1026.991,-23.344,-92.289,167.433,45.626,158.416
C08748=1026.985,-23.593,-92.275,167.431,45.628,158.416
C08749=1026.979,-23.843,-92.263,167.428,45.630,158.416
C08750=1026.973,-24.093,-92.249,167.426,45.632,158.417
C08751=1026.967,-24.342,-92.236,167.422,45.635,158.417
C08752=1026.961,-24.592,-92.222,167.420,45.637,158.417
C08753=1026.954,-24.841,-92.209,167.417,45.639,158.417
C08754=1026.949,-25.091,-92.196,167.415,45.641,158.417
C08755=1026.942,-25.341,-92.183,167.412,45.644,158.417
C08756=1026.936,-25.590,-92.170,167.409,45.646,158.417
C08757=1026.931,-25.839,-92.156,167.406,45.648,158.418
C08758=1026.924,-26.089,-92.142,167.404,45.651,158.418
C08759=1026.918,-26.339,-92.129,167.401,45.653,158.418
C08760=1026.912,-26.589,-92.116,167.398,45.655,158.418
C08761=1026.906,-26.838,-92.102,167.396,45.658,158.418
C08762=1026.900,-27.088,-92.090,167.393,45.660,158.418
C08763=1026.894,-27.337,-92.077,167.390,45.662,158.418
C08764=1026.888,-27.586,-92.063,167.387,45.665,158.418
C08765=1026.882,-27.836,-92.051,167.385,45.667,158.419
C08766=1026.876,-28.086,-92.037,167.381,45.670,158.419
C08767=1026.870,-28.335,-92.024,167.379,45.672,158.419
C08768=1026.863,-28.586,-92.011,167.377,45.675,158.419
C08769=1026.857,-28.835,-91.998,167.374,45.677,158.419
C08770=1026.851,-29.085,-91.985,167.371,45.680,158.419
C08771=1026.845,-29.334,-91.972,167.368,45.682,158.419
C08772=1026.839,-29.584,-91.960,167.366,45.685,158.420
C08773=1026.833,-29.833,-91.946,167.362,45.687,158.420
C08774=1026.827,-30.083,-91.934,167.360,45.690,158.420
C08775=1026.820,-30.332,-91.921,167.357,45.692,158.420
C08776=1026.814,-30.581,-91.907,167.354,45.695,158.420
C08777=1026.808,-30.831,-91.895,167.351,45.697,158.420
C08778=1026.801,-31.080,-91.882,167.349,45.699,158.421
C08779=1026.795,-31.330,-91.869,167.346,45.702,158.421
C08780=1026.789,-31.579,-91.856,167.343,45.704,158.421
C08781=1026.783,-31.830,-91.843,167.341,45.707,158.421
C08782=1026.777,-32.079,-91.830,167.337,45.709,158.421
C08783=1026.771,-32.329,-91.817,167.335,45.712,158.421
C08784=1026.765,-32.579,-91.805,167.333,45.714,158.421
C08785=1026.759,-32.828,-91.792,167.330,45.716,158.421
C08786=1026.753,-33.078,-91.779,167.327,45.719,158.422
C08787=1026.746,-33.327,-91.766,167.324,45.721,158.422
C08788=1026.741,-33.577,-91.753,167.322,45.723,158.422
C08789=1026.734,-33.827,-91.740,167.318,45.726,158.422
C08790=1026.728,-34.077,-91.727,167.316,45.728,158.422
C08791=1026.722,-34.326,-91.715,167.313,45.731,158.422
C08792=1026.716,-34.576,-91.702,167.310,45.733,158.422
C08793=1026.710,-34.826,-91.689,167.308,45.736,158.423
C08794=1026.703,-35.074,-91.676,167.305,45.738,158.423
C08795=1026.697,-35.324,-91.664,167.301,45.740,158.423
C08796=1026.692,-35.574,-91.652,167.299,45.743,158.423
C08797=1026.686,-35.823,-91.638,167.297,45.745,158.423
C08798=1026.680,-36.073,-91.626,167.293,45.748,158.423
C08799=1026.673,-36.353,-91.611,167.291,45.750,158.423
C08800=1026.666,-36.633,-91.597,167.287,45.753,158.423
C08801=1026.660,-36.913,-91.583,167.284,45.756,158.424
C08802=1026.653,-37.194,-91.568,167.282,45.759,158.424
C08803=1026.647,-37.443,-91.555,167.278,45.761,158.424
C08804=1026.641,-37.693,-91.543,167.276,45.763,158.424
C08805=1026.635,-37.942,-91.531,167.273,45.766,158.424
C08806=1026.629,-38.191,-91.518,167.270,45.768,158.424
C08807=1026.623,-38.441,-91.505,167.267,45.771,158.424
C08808=1026.617,-38.691,-91.493,167.265,45.773,158.425
C08809=1026.611,-38.940,-91.480,167.261,45.775,158.425
C08810=1026.605,-39.190,-91.467,167.259,45.778,158.425
C08811=1026.599,-39.440,-91.454,167.257,45.780,158.425
C08812=1026.592,-39.689,-91.442,167.253,45.783,158.425
C08813=1026.586,-39.939,-91.430,167.251,45.785,158.425
C08814=1026.580,-40.189,-91.417,167.247,45.788,158.425
C08815=1026.574,-40.439,-91.405,167.245,45.791,158.426
C08816=1026.568,-40.688,-91.393,167.242,45.793,158.426
C08817=1026.562,-40.937,-91.380,167.239,45.796,158.426
C08818=1026.555,-41.187,-91.368,167.237,45.798,158.426
C08819=1026.550,-41.436,-91.355,167.233,45.801,158.426
C08820=1026.544,-41.686,-91.343,167.231,45.803,158.426
C08821=1026.537,-41.936,-91.331,167.228,45.806,158.426
C08822=1026.531,-42.186,-91.318,167.225,45.808,158.426
C08823=1026.525,-42.435,-91.307,167.223,45.811,158.427
C08824=1026.519,-42.685,-91.294,167.220,45.813,158.427
C08825=1026.513,-42.934,-91.282,167.217,45.816,158.427
C08826=1026.507,-43.184,-91.270,167.214,45.818,158.427
C08827=1026.501,-43.434,-91.257,167.211,45.821,158.427
C08828=1026.495,-43.684,-91.244,167.208,45.823,158.427
C08829=1026.489,-43.933,-91.233,167.206,45.825,158.428
C08830=1026.483,-44.183,-91.220,167.202,45.828,158.428
C08831=1026.477,-44.432,-91.208,167.200,45.830,158.428
C08832=1026.470,-44.682,-91.196,167.197,45.833,158.428
C08833=1026.464,-44.932,-91.183,167.194,45.835,158.428
C08834=1026.458,-45.181,-91.172,167.192,45.837,158.428
C08835=1026.452,-45.431,-91.159,167.188,45.840,158.428
C08836=1026.447,-45.680,-91.147,167.186,45.842,158.428
C08837=1026.440,-45.930,-91.135,167.183,45.845,158.429
C08838=1026.435,-46.179,-91.122,167.180,45.847,158.429
C08839=1026.429,-46.429,-91.110,167.178,45.850,158.429
C08840=1026.422,-46.679,-91.098,167.174,45.853,158.429
C08841=1026.416,-46.929,-91.085,167.172,45.855,158.429
C08842=1026.410,-47.177,-91.074,167.169,45.857,158.429
C08843=1026.404,-47.427,-91.061,167.166,45.860,158.429
C08844=1026.398,-47.677,-91.049,167.163,45.862,158.429
C08845=1026.392,-47.927,-91.037,167.160,45.865,158.430
C08846=1026.386,-48.176,-91.025,167.158,45.867,158.430
C08847=1026.381,-48.426,-91.013,167.155,45.870,158.430
C08848=1026.374,-48.676,-91.001,167.152,45.872,158.430
C08849=1026.369,-48.925,-90.989,167.149,45.874,158.430
C08850=1026.362,-49.175,-90.977,167.146,45.877,158.430
C08851=1026.356,-49.425,-90.964,167.143,45.879,158.430
C08852=1026.351,-49.674,-90.952,167.141,45.882,158.431
C08853=1026.344,-49.923,-90.940,167.137,45.885,158.431
C08854=1026.339,-50.174,-90.928,167.135,45.887,158.431
C08855=1026.332,-50.424,-90.916,167.133,45.889,158.431
C08856=1026.327,-50.673,-90.904,167.129,45.892,158.431
C08857=1026.320,-50.922,-90.892,167.127,45.894,158.431
C08858=1026.314,-51.173,-90.880,167.123,45.897,158.431
C08859=1026.308,-51.422,-90.868,167.121,45.900,158.431
C08860=1026.302,-51.671,-90.857,167.117,45.902,158.431
C08861=1026.295,-51.921,-90.845,167.115,45.905,158.432
C08862=1026.290,-52.171,-90.833,167.112,45.908,158.432
C08863=1026.283,-52.452,-90.820,167.109,45.911,158.432
C08864=1026.275,-52.732,-90.807,167.105,45.914,158.432
C08865=1026.269,-53.012,-90.794,167.102,45.917,158.432
C08866=1026.262,-53.293,-90.780,167.099,45.920,158.433
C08867=1026.256,-53.542,-90.769,167.096,45.922,158.433
C08868=1026.250,-53.792,-90.758,167.093,45.925,158.433
C08869=1026.243,-54.042,-90.746,167.090,45.928,158.433
C08870=1026.238,-54.291,-90.734,167.087,45.930,158.433
C08871=1026.231,-54.541,-90.722,167.085,45.933,158.433
C08872=1026.225,-54.791,-90.711,167.081,45.936,158.433
C08873=1026.219,-55.040,-90.699,167.079,45.938,158.433
C08874=1026.212,-55.290,-90.687,167.075,45.941,158.434
C08875=1026.207,-55.539,-90.676,167.073,45.944,158.434
C08876=1026.201,-55.789,-90.664,167.070,45.946,158.434
C08877=1026.194,-56.039,-90.653,167.067,45.949,158.434
C08878=1026.188,-56.288,-90.641,167.064,45.952,158.434
C08879=1026.182,-56.538,-90.630,167.061,45.954,158.434
C08880=1026.177,-56.787,-90.618,167.058,45.957,158.435
C08881=1026.170,-57.038,-90.606,167.056,45.959,158.435
C08882=1026.164,-57.287,-90.595,167.052,45.962,158.435
C08883=1026.158,-57.537,-90.584,167.050,45.965,158.435
C08884=1026.152,-57.787,-90.572,167.047,45.967,158.435
C08885=1026.146,-58.036,-90.560,167.044,45.970,158.435
C08886=1026.140,-58.286,-90.549,167.041,45.973,158.435
C08887=1026.134,-58.535,-90.537,167.038,45.975,158.436
C08888=1026.128,-58.785,-90.526,167.035,45.978,158.436
C08889=1026.122,-59.034,-90.515,167.033,45.980,158.436
C08890=1026.116,-59.285,-90.503,167.029,45.983,158.436
C08891=1026.110,-59.534,-90.492,167.027,45.985,158.436
C08892=1026.104,-59.784,-90.480,167.023,45.988,158.436
C08893=1026.098,-60.033,-90.469,167.021,45.990,158.436
C08894=1026.091,-60.283,-90.457,167.018,45.993,158.437
C08895=1026.086,-60.533,-90.446,167.015,45.996,158.437
C08896=1026.080,-60.783,-90.434,167.012,45.999,158.437
C08897=1026.074,-61.032,-90.423,167.009,46.001,158.437
C08898=1026.067,-61.282,-90.411,167.007,46.003,158.437
C08899=1026.062,-61.531,-90.401,167.004,46.006,158.437
C08900=1026.056,-61.781,-90.388,167.001,46.009,158.437
C08901=1026.050,-62.031,-90.377,166.998,46.011,158.437
C08902=1026.044,-62.280,-90.366,166.995,46.014,158.438
C08903=1026.038,-62.530,-90.355,166.992,46.016,158.438
C08904=1026.032,-62.779,-90.343,166.990,46.019,158.438
C08905=1026.026,-63.029,-90.332,166.986,46.022,158.438
C08906=1026.021,-63.279,-90.321,166.984,46.024,158.438
C08907=1026.014,-63.529,-90.309,166.980,46.027,158.438
C08908=1026.008,-63.778,-90.298,166.978,46.029,158.438
C08909=1026.002,-64.028,-90.287,166.975,46.032,158.439
C08910=1025.996,-64.278,-90.276,166.972,46.034,158.439
C08911=1025.990,-64.527,-90.264,166.969,46.037,158.439
C08912=1025.984,-64.777,-90.252,166.966,46.040,158.439
C08913=1025.979,-65.027,-90.241,166.963,46.042,158.439
C08914=1025.973,-65.276,-90.231,166.961,46.045,158.439
C08915=1025.967,-65.527,-90.219,166.957,46.048,158.439
C08916=1025.961,-65.775,-90.208,166.955,46.050,158.439
C08917=1025.955,-66.025,-90.197,166.951,46.053,158.439
C08918=1025.948,-66.275,-90.186,166.949,46.055,158.440
C08919=1025.943,-66.525,-90.174,166.946,46.058,158.440
///RCONF 1,0,0,1,0,0,0,0,0,0,0,0,0,0,0,0,0,0,0,0,0,0,0,0
C08920=1025.938,-66.774,-90.163,166.943,46.060,158.440
C08921=1025.931,-67.025,-90.152,166.940,46.063,158.440
C08922=1025.925,-67.273,-90.140,166.937,46.065,158.440
C08923=1025.920,-67.523,-90.130,166.934,46.068,158.440
C08924=1025.913,-67.773,-90.118,166.931,46.071,158.440
C08925=1025.908,-68.023,-90.107,166.928,46.074,158.441
C08926=1025.903,-68.272,-90.096,166.925,46.076,158.441
C08927=1025.896,-68.554,-90.084,166.922,46.079,158.441
C08928=1025.889,-68.835,-90.071,166.919,46.082,158.441
C08929=1025.882,-69.117,-90.059,166.915,46.085,158.441
C08930=1025.876,-69.399,-90.046,166.912,46.088,158.441
C08931=1025.870,-69.649,-90.035,166.909,46.090,158.441
C08932=1025.864,-69.899,-90.024,166.906,46.093,158.441
C08933=1025.858,-70.148,-90.013,166.903,46.095,158.441
C08934=1025.852,-70.397,-90.001,166.900,46.098,158.442
C08935=1025.846,-70.647,-89.990,166.897,46.100,158.442
C08936=1025.840,-70.897,-89.979,166.895,46.103,158.442
C08937=1025.835,-71.147,-89.968,166.891,46.106,158.442
C08938=1025.830,-71.396,-89.957,166.889,46.108,158.442
C08939=1025.823,-71.646,-89.946,166.885,46.111,158.442
C08940=1025.817,-71.896,-89.935,166.883,46.113,158.442
C08941=1025.812,-72.145,-89.924,166.880,46.116,158.443
C08942=1025.806,-72.395,-89.913,166.877,46.118,158.443
C08943=1025.800,-72.644,-89.902,166.874,46.121,158.443
C08944=1025.794,-72.895,-89.892,166.871,46.123,158.443
C08945=1025.788,-73.145,-89.881,166.868,46.126,158.443
C08946=1025.783,-73.394,-89.869,166.865,46.128,158.443
C08947=1025.778,-73.644,-89.858,166.862,46.131,158.443
C08948=1025.771,-73.894,-89.847,166.859,46.133,158.443
C08949=1025.766,-74.143,-89.836,166.856,46.136,158.443
C08950=1025.760,-74.393,-89.825,166.854,46.138,158.444
C08951=1025.754,-74.642,-89.814,166.850,46.141,158.444
C08952=1025.749,-74.893,-89.804,166.848,46.144,158.444
C08953=1025.742,-75.142,-89.794,166.844,46.146,158.444
C08954=1025.736,-75.392,-89.783,166.842,46.149,158.444
C08955=1025.730,-75.641,-89.772,166.839,46.152,158.444
C08956=1025.724,-75.891,-89.761,166.835,46.155,158.444
C08957=1025.719,-76.141,-89.751,166.833,46.157,158.445
C08958=1025.713,-76.391,-89.740,166.830,46.160,158.445
C08959=1025.706,-76.640,-89.729,166.827,46.162,158.445
C08960=1025.700,-76.890,-89.718,166.824,46.165,158.445
C08961=1025.695,-77.140,-89.708,166.822,46.168,158.445
C08962=1025.689,-77.390,-89.697,166.818,46.171,158.445
C08963=1025.684,-77.639,-89.687,166.815,46.174,158.445
C08964=1025.677,-77.889,-89.677,166.812,46.176,158.445
C08965=1025.672,-78.138,-89.666,166.809,46.179,158.445
C08966=1025.666,-78.388,-89.655,166.807,46.181,158.446
C08967=1025.660,-78.638,-89.645,166.803,46.184,158.446
C08968=1025.654,-78.888,-89.634,166.801,46.187,158.446
C08969=1025.648,-79.137,-89.624,166.797,46.190,158.446
C08970=1025.642,-79.387,-89.613,166.794,46.193,158.446
C08971=1025.636,-79.637,-89.602,166.792,46.195,158.446
C08972=1025.631,-79.886,-89.592,166.788,46.198,158.446
C08973=1025.625,-80.136,-89.581,166.786,46.200,158.447
C08974=1025.619,-80.386,-89.571,166.783,46.203,158.447
C08975=1025.613,-80.636,-89.561,166.779,46.206,158.447
C08976=1025.607,-80.885,-89.551,166.777,46.209,158.447
C08977=1025.601,-81.135,-89.541,166.773,46.212,158.447
C08978=1025.594,-81.385,-89.530,166.770,46.215,158.447
C08979=1025.589,-81.635,-89.520,166.768,46.217,158.448
C08980=1025.583,-81.885,-89.509,166.765,46.220,158.448
C08981=1025.577,-82.134,-89.499,166.762,46.222,158.448
C08982=1025.571,-82.384,-89.488,166.759,46.225,158.448
C08983=1025.565,-82.634,-89.479,166.755,46.228,158.448
C08984=1025.559,-82.883,-89.468,166.753,46.231,158.448
C08985=1025.553,-83.133,-89.458,166.750,46.234,158.448
C08986=1025.547,-83.382,-89.448,166.747,46.237,158.449
C08987=1025.541,-83.632,-89.438,166.744,46.239,158.449
C08988=1025.536,-83.882,-89.428,166.741,46.242,158.449
C08989=1025.529,-84.131,-89.418,166.737,46.245,158.449
C08990=1025.524,-84.382,-89.407,166.735,46.248,158.449
C08991=1025.517,-84.665,-89.396,166.732,46.251,158.449
C08992=1025.511,-84.948,-89.384,166.727,46.254,158.449
C08993=1025.503,-85.233,-89.373,166.724,46.258,158.450
C08994=1025.497,-85.517,-89.361,166.721,46.261,158.450
C08995=1025.491,-85.767,-89.352,166.719,46.263,158.450
C08996=1025.485,-86.016,-89.341,166.715,46.266,158.450
C08997=1025.480,-86.266,-89.331,166.712,46.269,158.450
C08998=1025.474,-86.516,-89.321,166.710,46.272,158.450
C08999=1025.468,-86.765,-89.310,166.706,46.275,158.451
C09000=1025.462,-87.015,-89.301,166.703,46.277,158.451
C09001=1025.456,-87.265,-89.290,166.701,46.280,158.451
